LIN {X 0,Y 524.038,Z 318.828,A -85,B 0,C 180,E1 -4863.075,E2 -4863.075} C_VEL
LIN {X 0,Y 524.003,Z 318.833,A -85,B 0,C 180,E1 -4866.16,E2 -4866.16} C_VEL
LIN {X 0,Y 523.983,Z 318.838,A -85,B 0,C 180,E1 -4869.262,E2 -4869.262} C_VEL
LIN {X 0,Y 524.003,Z 318.838,A -85,B 0,C 180,E1 -4871.736,E2 -4871.736} C_VEL
LIN {X 0,Y 523.989,Z 318.836,A -85,B 0,C 180,E1 -4875.048,E2 -4875.048} C_VEL
LIN {X 0,Y 523.917,Z 318.849,A -85,B 0,C 180,E1 -4877.971,E2 -4877.971} C_VEL
LIN {X 0,Y 523.92,Z 318.841,A -85,B 0,C 180,E1 -4880.412,E2 -4880.412} C_VEL
LIN {X 0,Y 523.889,Z 318.848,A -85,B 0,C 180,E1 -4882.895,E2 -4882.895} C_VEL
LIN {X 0,Y 523.902,Z 318.85,A -85,B 0,C 180,E1 -4885.422,E2 -4885.422} C_VEL
LIN {X 0,Y 523.9,Z 318.847,A -85,B 0,C 180,E1 -4888.003,E2 -4888.003} C_VEL
LIN {X 0,Y 523.901,Z 318.839,A -85,B 0,C 180,E1 -4890.846,E2 -4890.846} C_VEL
LIN {X 0,Y 523.929,Z 318.847,A -85,B 0,C 180,E1 -4893.729,E2 -4893.729} C_VEL
LIN {X 0,Y 523.861,Z 318.844,A -85,B 0,C 180,E1 -4896.394,E2 -4896.394} C_VEL
LIN {X 0,Y 523.889,Z 318.852,A -85,B 0,C 180,E1 -4899.088,E2 -4899.088} C_VEL
LIN {X 0,Y 523.889,Z 318.848,A -85,B 0,C 180,E1 -4902.126,E2 -4902.126} C_VEL
LIN {X 0,Y 523.931,Z 318.847,A -85,B 0,C 180,E1 -4905.312,E2 -4905.312} C_VEL
LIN {X 0,Y 523.872,Z 318.851,A -85,B 0,C 180,E1 -4906.869,E2 -4906.869} C_VEL
LIN {X 0,Y 523.182,Z 318.943,A -85,B 0,C 180,E1 -4907.51,E2 -4907.51} C_VEL
LIN {X 0,Y 520.313,Z 319.296,A -85,B 0,C 180,E1 -4908.552,E2 -4908.552} C_VEL
LIN {X 0,Y 517.911,Z 319.598,A -85,B 0,C 180,E1 -4909.39,E2 -4909.39} C_VEL
LIN {X 0,Y 516.897,Z 319.721,A -85,B 0,C 180,E1 -4910.038,E2 -4910.038} C_VEL
LIN {X 0,Y 516.823,Z 319.729,A -85,B 0,C 180,E1 -4910.257,E2 -4910.257} C_VEL
LIN {X 0,Y 516.799,Z 319.74,A -85,B 0,C 180,E1 -4913.247,E2 -4913.247} C_VEL
LIN {X 0,Y 516.869,Z 319.723,A -85,B 0,C 180,E1 -4916.117,E2 -4916.117} C_VEL
LIN {X 0,Y 516.852,Z 319.731,A -85,B 0,C 180,E1 -4918.944,E2 -4918.944} C_VEL
LIN {X 0,Y 516.878,Z 319.819,A -85,B 0,C 180,E1 -4922.214,E2 -4922.214} C_VEL
LIN {X 0,Y 518.337,Z 327.517,A -85,B 0,C 180,E1 -4923.638,E2 -4923.638} C_VEL
LIN {X 0,Y 517.957,Z 343.652,A -85,B 0,C 180,E1 -4926.406,E2 -4926.406} C_VEL
LIN {X 0,Y 518.607,Z 346.948,A -85,B 0,C 180,E1 -4926.504,E2 -4926.504} C_VEL
LIN {X 0,Y 520.476,Z 356.835,A -85,B 0,C 180,E1 -4926.715,E2 -4926.715} C_VEL
LIN {X 0,Y 519.751,Z 479.979,A -85,B 0,C 180,E1 -4928.457,E2 -4928.457} C_VEL
LIN {X 0,Y 519.484,Z 494.208,A -85,B 0,C 180,E1 -4928.809,E2 -4928.809} C_VEL
LIN {X 0,Y 519.165,Z 508.132,A -85,B 0,C 180,E1 -4929.319,E2 -4929.319} C_VEL
LIN {X 0,Y 518.806,Z 521.885,A -85,B 0,C 180,E1 -4929.998,E2 -4929.998} C_VEL
LIN {X 0,Y 518.35,Z 534.66,A -85,B 0,C 180,E1 -4930.804,E2 -4930.804} C_VEL
LIN {X 0,Y 517.995,Z 545.305,A -85,B 0,C 180,E1 -4931.633,E2 -4931.633} C_VEL
LIN {X 0,Y 517.56,Z 555.862,A -85,B 0,C 180,E1 -4932.618,E2 -4932.618} C_VEL
LIN {X 0,Y 517.214,Z 566.524,A -85,B 0,C 180,E1 -4933.826,E2 -4933.826} C_VEL
LIN {X 0,Y 516.89,Z 575.271,A -85,B 0,C 180,E1 -4935.028,E2 -4935.028} C_VEL
LIN {X 0,Y 516.643,Z 583.607,A -85,B 0,C 180,E1 -4936.429,E2 -4936.429} C_VEL
LIN {X 0,Y 516.481,Z 590.258,A -85,B 0,C 180,E1 -4937.824,E2 -4937.824} C_VEL
LIN {X 0,Y 516.386,Z 594.836,A -85,B 0,C 180,E1 -4939.016,E2 -4939.016} C_VEL
LIN {X 0,Y 516.303,Z 598.458,A -85,B 0,C 180,E1 -4940.203,E2 -4940.203} C_VEL
LIN {X 0,Y 516.257,Z 601.259,A -85,B 0,C 180,E1 -4941.388,E2 -4941.388} C_VEL
LIN {X 0,Y 516.284,Z 603.699,A -85,B 0,C 180,E1 -4942.963,E2 -4942.963} C_VEL
LIN {X 0,Y 516.271,Z 604.789,A -85,B 0,C 180,E1 -4944.532,E2 -4944.532} C_VEL
LIN {X 0,Y 516.293,Z 604.557,A -85,B 0,C 180,E1 -4946.097,E2 -4946.097} C_VEL
LIN {X 0,Y 516.259,Z 603.009,A -85,B 0,C 180,E1 -4947.659,E2 -4947.659} C_VEL
LIN {X 0,Y 516.172,Z 600.122,A -85,B 0,C 180,E1 -4949.22,E2 -4949.22} C_VEL
LIN {X 0,Y 516.248,Z 595.813,A -85,B 0,C 180,E1 -4950.78,E2 -4950.78} C_VEL
LIN {X 0,Y 516.372,Z 589.959,A -85,B 0,C 180,E1 -4952.34,E2 -4952.34} C_VEL
LIN {X 0,Y 516.636,Z 583.37,A -85,B 0,C 180,E1 -4953.705,E2 -4953.705} C_VEL
LIN {X 0,Y 516.969,Z 575.193,A -85,B 0,C 180,E1 -4955.07,E2 -4955.07} C_VEL
LIN {X 0,Y 517.262,Z 566.698,A -85,B 0,C 180,E1 -4956.24,E2 -4956.24} C_VEL
LIN {X 0,Y 517.567,Z 556.458,A -85,B 0,C 180,E1 -4957.409,E2 -4957.409} C_VEL
LIN {X 0,Y 517.997,Z 544.966,A -85,B 0,C 180,E1 -4958.485,E2 -4958.485} C_VEL
LIN {X 0,Y 518.378,Z 533.526,A -85,B 0,C 180,E1 -4959.363,E2 -4959.363} C_VEL
LIN {X 0,Y 518.787,Z 520.975,A -85,B 0,C 180,E1 -4960.143,E2 -4960.143} C_VEL
LIN {X 0,Y 519.171,Z 507.994,A -85,B 0,C 180,E1 -4960.777,E2 -4960.777} C_VEL
LIN {X 0,Y 519.532,Z 493.96,A -85,B 0,C 180,E1 -4961.287,E2 -4961.287} C_VEL
LIN {X 0,Y 519.706,Z 480.239,A -85,B 0,C 180,E1 -4961.629,E2 -4961.629} C_VEL
LIN {X 0,Y 520.413,Z 355.748,A -85,B 0,C 180,E1 -4963.392,E2 -4963.392} C_VEL
LIN {X 0,Y 517.973,Z 343.725,A -85,B 0,C 180,E1 -4963.666,E2 -4963.666} C_VEL
LIN {X 0,Y 518.387,Z 328.115,A -85,B 0,C 180,E1 -4966.339,E2 -4966.339} C_VEL
LIN {X 0,Y 517.157,Z 321.108,A -85,B 0,C 180,E1 -4967.626,E2 -4967.626} C_VEL
LIN {X 0,Y 516.889,Z 319.725,A -85,B 0,C 180,E1 -4967.934,E2 -4967.934} C_VEL
LIN {X 0,Y 516.881,Z 319.729,A -85,B 0,C 180,E1 -4970.703,E2 -4970.703} C_VEL
LIN {X 0,Y 516.853,Z 319.73,A -85,B 0,C 180,E1 -4973.225,E2 -4973.225} C_VEL
LIN {X 0,Y 516.858,Z 319.726,A -85,B 0,C 180,E1 -4976.176,E2 -4976.176} C_VEL
LIN {X 0,Y 516.831,Z 319.731,A -85,B 0,C 180,E1 -4978.421,E2 -4978.421} C_VEL
LIN {X 0,Y 516.851,Z 319.73,A -85,B 0,C 180,E1 -4981.112,E2 -4981.112} C_VEL
LIN {X 0,Y 516.868,Z 319.723,A -85,B 0,C 180,E1 -4983.958,E2 -4983.958} C_VEL
LIN {X 0,Y 516.799,Z 319.738,A -85,B 0,C 180,E1 -4986.753,E2 -4986.753} C_VEL
LIN {X 0,Y 516.831,Z 319.726,A -85,B 0,C 180,E1 -4989.726,E2 -4989.726} C_VEL
LIN {X 0,Y 516.84,Z 319.732,A -85,B 0,C 180,E1 -4992.836,E2 -4992.836} C_VEL
LIN {X 0,Y 516.9,Z 319.721,A -85,B 0,C 180,E1 -4995.007,E2 -4995.007} C_VEL
LIN {X 0,Y 516.833,Z 319.732,A -85,B 0,C 180,E1 -4998.409,E2 -4998.409} C_VEL
LIN {X 0,Y 516.856,Z 319.724,A -85,B 0,C 180,E1 -5001.281,E2 -5001.281} C_VEL
LIN {X 0,Y 516.853,Z 319.731,A -85,B 0,C 180,E1 -5004.673,E2 -5004.673} C_VEL
LIN {X 0,Y 516.871,Z 319.718,A -85,B 0,C 180,E1 -5007.462,E2 -5007.462} C_VEL
LIN {X 0,Y 516.848,Z 319.732,A -85,B 0,C 180,E1 -5010.49,E2 -5010.49} C_VEL
LIN {X 0,Y 516.84,Z 319.723,A -85,B 0,C 180,E1 -5013.337,E2 -5013.337} C_VEL
LIN {X 0,Y 516.884,Z 319.723,A -85,B 0,C 180,E1 -5015.926,E2 -5015.926} C_VEL
LIN {X 0,Y 516.869,Z 319.721,A -85,B 0,C 180,E1 -5018.461,E2 -5018.461} C_VEL
LIN {X 0,Y 516.883,Z 319.717,A -85,B 0,C 180,E1 -5020.954,E2 -5020.954} C_VEL
LIN {X 0,Y 516.835,Z 319.726,A -85,B 0,C 180,E1 -5023.407,E2 -5023.407} C_VEL
LIN {X 0,Y 516.877,Z 319.723,A -85,B 0,C 180,E1 -5025.833,E2 -5025.833} C_VEL
LIN {X 0,Y 516.952,Z 319.702,A -85,B 0,C 180,E1 -5029.028,E2 -5029.028} C_VEL
LIN {X 0,Y 516.947,Z 319.718,A -85,B 0,C 180,E1 -5032.186,E2 -5032.186} C_VEL
LIN {X 0,Y 516.991,Z 319.71,A -85,B 0,C 180,E1 -5034.539,E2 -5034.539} C_VEL
LIN {X 0,Y 517.081,Z 319.697,A -85,B 0,C 180,E1 -5037.663,E2 -5037.663} C_VEL
LIN {X 0,Y 517.093,Z 319.692,A -85,B 0,C 180,E1 -5040.779,E2 -5040.779} C_VEL
LIN {X 0,Y 516.951,Z 319.711,A -85,B 0,C 180,E1 -5043.117,E2 -5043.117} C_VEL
LIN {X 0,Y 516.978,Z 319.713,A -85,B 0,C 180,E1 -5046.243,E2 -5046.243} C_VEL
LIN {X 0,Y 516.941,Z 319.714,A -85,B 0,C 180,E1 -5049.389,E2 -5049.389} C_VEL
LIN {X 0,Y 516.956,Z 319.717,A -85,B 0,C 180,E1 -5051.807,E2 -5051.807} C_VEL
LIN {X 0,Y 516.949,Z 319.711,A -85,B 0,C 180,E1 -5055.146,E2 -5055.146} C_VEL
LIN {X 0,Y 516.916,Z 319.719,A -85,B 0,C 180,E1 -5058.222,E2 -5058.222} C_VEL
LIN {X 0,Y 516.916,Z 319.716,A -85,B 0,C 180,E1 -5060.701,E2 -5060.701} C_VEL
LIN {X 0,Y 516.893,Z 319.724,A -85,B 0,C 180,E1 -5064.073,E2 -5064.073} C_VEL
LIN {X 0,Y 516.914,Z 319.716,A -85,B 0,C 180,E1 -5066.658,E2 -5066.658} C_VEL
LIN {X 0,Y 516.913,Z 319.722,A -85,B 0,C 180,E1 -5069.523,E2 -5069.523} C_VEL
LIN {X 0,Y 516.898,Z 319.718,A -85,B 0,C 180,E1 -5072.543,E2 -5072.543} C_VEL
LIN {X 0,Y 516.871,Z 319.727,A -85,B 0,C 180,E1 -5075.33,E2 -5075.33} C_VEL
LIN {X 0,Y 516.881,Z 319.725,A -85,B 0,C 180,E1 -5077.943,E2 -5077.943} C_VEL
LIN {X 0,Y 516.885,Z 319.721,A -85,B 0,C 180,E1 -5080.741,E2 -5080.741} C_VEL
LIN {X 0,Y 516.884,Z 319.721,A -85,B 0,C 180,E1 -5082.831,E2 -5082.831} C_VEL
LIN {X 0,Y 516.897,Z 319.721,A -85,B 0,C 180,E1 -5085.007,E2 -5085.007} C_VEL
LIN {X 0,Y 516.915,Z 319.717,A -85,B 0,C 180,E1 -5088.399,E2 -5088.399} C_VEL
LIN {X 0,Y 516.882,Z 319.728,A -85,B 0,C 180,E1 -5091.284,E2 -5091.284} C_VEL
LIN {X 0,Y 516.89,Z 319.722,A -85,B 0,C 180,E1 -5094.221,E2 -5094.221} C_VEL
LIN {X 0,Y 516.897,Z 319.725,A -85,B 0,C 180,E1 -5097.053,E2 -5097.053} C_VEL
LIN {X 0,Y 516.894,Z 319.724,A -85,B 0,C 180,E1 -5099.796,E2 -5099.796} C_VEL
LIN {X 0,Y 516.928,Z 319.718,A -85,B 0,C 180,E1 -5102.467,E2 -5102.467} C_VEL
LIN {X 0,Y 516.962,Z 319.819,A -85,B 0,C 180,E1 -5103.83,E2 -5103.83} C_VEL
LIN {X 0,Y 519.173,Z 330.998,A -85,B 0,C 180,E1 -5105.614,E2 -5105.614} C_VEL
LIN {X 0,Y 518.581,Z 350.939,A -85,B 0,C 180,E1 -5108.536,E2 -5108.536} C_VEL
LIN {X 0,Y 518.001,Z 370.708,A -85,B 0,C 180,E1 -5111.377,E2 -5111.377} C_VEL
LIN {X 0,Y 520.347,Z 384.922,A -85,B 0,C 180,E1 -5111.666,E2 -5111.666} C_VEL
LIN {X 0,Y 519.63,Z 509.015,A -85,B 0,C 180,E1 -5113.424,E2 -5113.424} C_VEL
LIN {X 0,Y 519.367,Z 523.324,A -85,B 0,C 180,E1 -5113.786,E2 -5113.786} C_VEL
LIN {X 0,Y 519.051,Z 536.906,A -85,B 0,C 180,E1 -5114.288,E2 -5114.288} C_VEL
LIN {X 0,Y 518.654,Z 550.881,A -85,B 0,C 180,E1 -5114.98,E2 -5114.98} C_VEL
LIN {X 0,Y 518.219,Z 563.384,A -85,B 0,C 180,E1 -5115.77,E2 -5115.77} C_VEL
LIN {X 0,Y 517.825,Z 574.814,A -85,B 0,C 180,E1 -5116.66,E2 -5116.66} C_VEL
LIN {X 0,Y 517.445,Z 585.278,A -85,B 0,C 180,E1 -5117.644,E2 -5117.644} C_VEL
LIN {X 0,Y 517.138,Z 595.771,A -85,B 0,C 180,E1 -5118.833,E2 -5118.833} C_VEL
LIN {X 0,Y 516.813,Z 604.395,A -85,B 0,C 180,E1 -5120.015,E2 -5120.015} C_VEL
LIN {X 0,Y 516.59,Z 612.657,A -85,B 0,C 180,E1 -5121.393,E2 -5121.393} C_VEL
LIN {X 0,Y 516.445,Z 618.44,A -85,B 0,C 180,E1 -5122.572,E2 -5122.572} C_VEL
LIN {X 0,Y 516.395,Z 623.18,A -85,B 0,C 180,E1 -5123.749,E2 -5123.749} C_VEL
LIN {X 0,Y 516.306,Z 627.019,A -85,B 0,C 180,E1 -5124.924,E2 -5124.924} C_VEL
LIN {X 0,Y 516.324,Z 629.978,A -85,B 0,C 180,E1 -5126.098,E2 -5126.098} C_VEL
LIN {X 0,Y 516.259,Z 632.685,A -85,B 0,C 180,E1 -5127.659,E2 -5127.659} C_VEL
LIN {X 0,Y 516.157,Z 634.024,A -85,B 0,C 180,E1 -5129.22,E2 -5129.22} C_VEL
LIN {X 0,Y 516.157,Z 634.024,A -85,B 0,C 180,E1 -5130.78,E2 -5130.78} C_VEL
LIN {X 0,Y 516.259,Z 632.686,A -85,B 0,C 180,E1 -5132.341,E2 -5132.341} C_VEL
LIN {X 0,Y 516.324,Z 629.98,A -85,B 0,C 180,E1 -5133.903,E2 -5133.903} C_VEL
LIN {X 0,Y 516.367,Z 625.828,A -85,B 0,C 180,E1 -5135.467,E2 -5135.467} C_VEL
LIN {X 0,Y 516.402,Z 620.109,A -85,B 0,C 180,E1 -5137.036,E2 -5137.036} C_VEL
LIN {X 0,Y 516.582,Z 613.665,A -85,B 0,C 180,E1 -5138.41,E2 -5138.41} C_VEL
LIN {X 0,Y 516.779,Z 605.659,A -85,B 0,C 180,E1 -5139.788,E2 -5139.788} C_VEL
LIN {X 0,Y 517.078,Z 597.288,A -85,B 0,C 180,E1 -5140.969,E2 -5140.969} C_VEL
LIN {X 0,Y 517.414,Z 586.88,A -85,B 0,C 180,E1 -5142.19,E2 -5142.19} C_VEL
LIN {X 0,Y 517.783,Z 575.973,A -85,B 0,C 180,E1 -5143.241,E2 -5143.241} C_VEL
LIN {X 0,Y 518.211,Z 563.369,A -85,B 0,C 180,E1 -5144.23,E2 -5144.23} C_VEL
LIN {X 0,Y 518.664,Z 550.862,A -85,B 0,C 180,E1 -5145.02,E2 -5145.02} C_VEL
LIN {X 0,Y 519.03,Z 538.006,A -85,B 0,C 180,E1 -5145.662,E2 -5145.662} C_VEL
LIN {X 0,Y 519.34,Z 524.353,A -85,B 0,C 180,E1 -5146.179,E2 -5146.179} C_VEL
LIN {X 0,Y 519.621,Z 510.128,A -85,B 0,C 180,E1 -5146.552,E2 -5146.552} C_VEL
LIN {X 0,Y 519.826,Z 481.992,A -85,B 0,C 180,E1 -5146.975,E2 -5146.975} C_VEL
LIN {X 0,Y 520.36,Z 383.971,A -85,B 0,C 180,E1 -5148.347,E2 -5148.347} C_VEL
LIN {X 0,Y 518.017,Z 370.538,A -85,B 0,C 180,E1 -5148.633,E2 -5148.633} C_VEL
LIN {X 0,Y 518.626,Z 349.478,A -85,B 0,C 180,E1 -5151.671,E2 -5151.671} C_VEL
LIN {X 0,Y 519.184,Z 330.985,A -85,B 0,C 180,E1 -5154.385,E2 -5154.385} C_VEL
LIN {X 0,Y 516.944,Z 319.769,A -85,B 0,C 180,E1 -5156.196,E2 -5156.196} C_VEL
LIN {X 0,Y 516.924,Z 319.717,A -85,B 0,C 180,E1 -5159.305,E2 -5159.305} C_VEL
LIN {X 0,Y 516.898,Z 319.725,A -85,B 0,C 180,E1 -5162.544,E2 -5162.544} C_VEL
LIN {X 0,Y 516.869,Z 319.724,A -85,B 0,C 180,E1 -5165.33,E2 -5165.33} C_VEL
LIN {X 0,Y 516.882,Z 319.723,A -85,B 0,C 180,E1 -5167.943,E2 -5167.943} C_VEL
LIN {X 0,Y 516.885,Z 319.725,A -85,B 0,C 180,E1 -5170.742,E2 -5170.742} C_VEL
LIN {X 0,Y 516.884,Z 319.723,A -85,B 0,C 180,E1 -5172.832,E2 -5172.832} C_VEL
LIN {X 0,Y 516.897,Z 319.72,A -85,B 0,C 180,E1 -5175.007,E2 -5175.007} C_VEL
LIN {X 0,Y 516.916,Z 319.723,A -85,B 0,C 180,E1 -5178.399,E2 -5178.399} C_VEL
LIN {X 0,Y 516.881,Z 319.72,A -85,B 0,C 180,E1 -5181.284,E2 -5181.284} C_VEL
LIN {X 0,Y 516.87,Z 319.727,A -85,B 0,C 180,E1 -5184.22,E2 -5184.22} C_VEL
LIN {X 0,Y 516.898,Z 319.718,A -85,B 0,C 180,E1 -5187.053,E2 -5187.053} C_VEL
LIN {X 0,Y 516.895,Z 319.721,A -85,B 0,C 180,E1 -5189.797,E2 -5189.797} C_VEL
LIN {X 0,Y 516.895,Z 319.723,A -85,B 0,C 180,E1 -5192.466,E2 -5192.466} C_VEL
LIN {X 0,Y 516.868,Z 319.722,A -85,B 0,C 180,E1 -5195.07,E2 -5195.07} C_VEL
LIN {X 0,Y 516.873,Z 319.722,A -85,B 0,C 180,E1 -5197.622,E2 -5197.622} C_VEL
LIN {X 0,Y 516.933,Z 319.723,A -85,B 0,C 180,E1 -5200.13,E2 -5200.13} C_VEL
LIN {X 0,Y 516.901,Z 319.719,A -85,B 0,C 180,E1 -5202.595,E2 -5202.595} C_VEL
LIN {X 0,Y 516.947,Z 319.712,A -85,B 0,C 180,E1 -5205.03,E2 -5205.03} C_VEL
LIN {X 0,Y 516.971,Z 319.715,A -85,B 0,C 180,E1 -5208.234,E2 -5208.234} C_VEL
LIN {X 0,Y 516.955,Z 319.711,A -85,B 0,C 180,E1 -5211.4,E2 -5211.4} C_VEL
LIN {X 0,Y 517.016,Z 319.705,A -85,B 0,C 180,E1 -5214.54,E2 -5214.54} C_VEL
LIN {X 0,Y 517.078,Z 319.697,A -85,B 0,C 180,E1 -5217.663,E2 -5217.663} C_VEL
LIN {X 0,Y 517.069,Z 319.703,A -85,B 0,C 180,E1 -5220,E2 -5220} C_VEL
LIN {X 0,Y 517.081,Z 319.697,A -85,B 0,C 180,E1 -5222.337,E2 -5222.337} C_VEL
LIN {X 0,Y 516.97,Z 319.708,A -85,B 0,C 180,E1 -5226.244,E2 -5226.244} C_VEL
LIN {X 0,Y 516.939,Z 319.717,A -85,B 0,C 180,E1 -5229.39,E2 -5229.39} C_VEL
LIN {X 0,Y 516.957,Z 319.716,A -85,B 0,C 180,E1 -5231.807,E2 -5231.807} C_VEL
LIN {X 0,Y 516.942,Z 319.715,A -85,B 0,C 180,E1 -5235.143,E2 -5235.143} C_VEL
LIN {X 0,Y 516.878,Z 319.723,A -85,B 0,C 180,E1 -5238.224,E2 -5238.224} C_VEL
LIN {X 0,Y 516.875,Z 319.718,A -85,B 0,C 180,E1 -5240.703,E2 -5240.703} C_VEL
LIN {X 0,Y 516.844,Z 319.729,A -85,B 0,C 180,E1 -5243.225,E2 -5243.225} C_VEL
LIN {X 0,Y 516.883,Z 319.722,A -85,B 0,C 180,E1 -5246.181,E2 -5246.181} C_VEL
LIN {X 0,Y 516.833,Z 319.724,A -85,B 0,C 180,E1 -5248.421,E2 -5248.421} C_VEL
LIN {X 0,Y 516.852,Z 319.719,A -85,B 0,C 180,E1 -5251.112,E2 -5251.112} C_VEL
LIN {X 0,Y 516.884,Z 319.722,A -85,B 0,C 180,E1 -5253.961,E2 -5253.961} C_VEL
LIN {X 0,Y 516.803,Z 319.724,A -85,B 0,C 180,E1 -5256.753,E2 -5256.753} C_VEL
LIN {X 0,Y 516.856,Z 319.729,A -85,B 0,C 180,E1 -5259.189,E2 -5259.189} C_VEL
LIN {X 0,Y 516.834,Z 319.729,A -85,B 0,C 180,E1 -5261.783,E2 -5261.783} C_VEL
LIN {X 0,Y 516.9,Z 319.723,A -85,B 0,C 180,E1 -5265.007,E2 -5265.007} C_VEL
LIN {X 0,Y 516.83,Z 319.729,A -85,B 0,C 180,E1 -5268.41,E2 -5268.41} C_VEL
LIN {X 0,Y 516.823,Z 319.729,A -85,B 0,C 180,E1 -5270.257,E2 -5270.257} C_VEL
LIN {X 0,Y 516.178,Z 319.815,A -85,B 0,C 180,E1 -5270.907,E2 -5270.907} C_VEL
LIN {X 0,Y 513.324,Z 320.171,A -85,B 0,C 180,E1 -5271.963,E2 -5271.963} C_VEL
LIN {X 0,Y 510.894,Z 320.475,A -85,B 0,C 180,E1 -5272.813,E2 -5272.813} C_VEL
LIN {X 0,Y 509.846,Z 320.604,A -85,B 0,C 180,E1 -5273.47,E2 -5273.47} C_VEL
LIN {X 0,Y 509.758,Z 320.612,A -85,B 0,C 180,E1 -5273.692,E2 -5273.692} C_VEL
LIN {X 0,Y 509.827,Z 320.601,A -85,B 0,C 180,E1 -5276.536,E2 -5276.536} C_VEL
LIN {X 0,Y 509.804,Z 320.609,A -85,B 0,C 180,E1 -5279.331,E2 -5279.331} C_VEL
LIN {X 0,Y 509.835,Z 320.687,A -85,B 0,C 180,E1 -5281.998,E2 -5281.998} C_VEL
LIN {X 0,Y 511.465,Z 329.337,A -85,B 0,C 180,E1 -5283.625,E2 -5283.625} C_VEL
LIN {X 0,Y 511.046,Z 343.971,A -85,B 0,C 180,E1 -5286.167,E2 -5286.167} C_VEL
LIN {X 0,Y 513.649,Z 356.408,A -85,B 0,C 180,E1 -5286.453,E2 -5286.453} C_VEL
LIN {X 0,Y 512.97,Z 480.449,A -85,B 0,C 180,E1 -5288.237,E2 -5288.237} C_VEL
LIN {X 0,Y 512.669,Z 494.537,A -85,B 0,C 180,E1 -5288.592,E2 -5288.592} C_VEL
LIN {X 0,Y 512.329,Z 508.352,A -85,B 0,C 180,E1 -5289.105,E2 -5289.105} C_VEL
LIN {X 0,Y 511.937,Z 520.818,A -85,B 0,C 180,E1 -5289.718,E2 -5289.718} C_VEL
LIN {X 0,Y 511.522,Z 533.849,A -85,B 0,C 180,E1 -5290.538,E2 -5290.538} C_VEL
LIN {X 0,Y 511.067,Z 545.623,A -85,B 0,C 180,E1 -5291.457,E2 -5291.457} C_VEL
LIN {X 0,Y 510.57,Z 557.352,A -85,B 0,C 180,E1 -5292.579,E2 -5292.579} C_VEL
LIN {X 0,Y 510.204,Z 567.776,A -85,B 0,C 180,E1 -5293.803,E2 -5293.803} C_VEL
LIN {X 0,Y 509.839,Z 576.337,A -85,B 0,C 180,E1 -5295.021,E2 -5295.021} C_VEL
LIN {X 0,Y 509.566,Z 584.47,A -85,B 0,C 180,E1 -5296.44,E2 -5296.44} C_VEL
LIN {X 0,Y 509.42,Z 590.175,A -85,B 0,C 180,E1 -5297.652,E2 -5297.652} C_VEL
LIN {X 0,Y 509.285,Z 596.116,A -85,B 0,C 180,E1 -5299.263,E2 -5299.263} C_VEL
LIN {X 0,Y 509.178,Z 599.541,A -85,B 0,C 180,E1 -5300.466,E2 -5300.466} C_VEL
LIN {X 0,Y 509.17,Z 602.756,A -85,B 0,C 180,E1 -5302.066,E2 -5302.066} C_VEL
LIN {X 0,Y 509.174,Z 604.57,A -85,B 0,C 180,E1 -5303.66,E2 -5303.66} C_VEL
LIN {X 0,Y 509.128,Z 605.055,A -85,B 0,C 180,E1 -5305.249,E2 -5305.249} C_VEL
LIN {X 0,Y 509.182,Z 604.219,A -85,B 0,C 180,E1 -5306.835,E2 -5306.835} C_VEL
LIN {X 0,Y 509.116,Z 602.063,A -85,B 0,C 180,E1 -5308.418,E2 -5308.418} C_VEL
LIN {X 0,Y 509.13,Z 598.535,A -85,B 0,C 180,E1 -5310,E2 -5310} C_VEL
LIN {X 0,Y 509.303,Z 594.935,A -85,B 0,C 180,E1 -5311.186,E2 -5311.186} C_VEL
LIN {X 0,Y 509.302,Z 590.439,A -85,B 0,C 180,E1 -5312.373,E2 -5312.373} C_VEL
LIN {X 0,Y 509.586,Z 583.925,A -85,B 0,C 180,E1 -5313.756,E2 -5313.756} C_VEL
LIN {X 0,Y 509.95,Z 575.857,A -85,B 0,C 180,E1 -5315.14,E2 -5315.14} C_VEL
LIN {X 0,Y 510.264,Z 567.451,A -85,B 0,C 180,E1 -5316.326,E2 -5316.326} C_VEL
LIN {X 0,Y 510.585,Z 557.063,A -85,B 0,C 180,E1 -5317.539,E2 -5317.539} C_VEL
LIN {X 0,Y 511.048,Z 545.971,A -85,B 0,C 180,E1 -5318.601,E2 -5318.601} C_VEL
LIN {X 0,Y 511.51,Z 533.299,A -85,B 0,C 180,E1 -5319.59,E2 -5319.59} C_VEL
LIN {X 0,Y 511.951,Z 520.646,A -85,B 0,C 180,E1 -5320.38,E2 -5320.38} C_VEL
LIN {X 0,Y 512.322,Z 507.526,A -85,B 0,C 180,E1 -5321.022,E2 -5321.022} C_VEL
LIN {X 0,Y 512.72,Z 493.202,A -85,B 0,C 180,E1 -5321.539,E2 -5321.539} C_VEL
LIN {X 0,Y 512.957,Z 478.712,A -85,B 0,C 180,E1 -5321.885,E2 -5321.885} C_VEL
LIN {X 0,Y 513.628,Z 356.48,A -85,B 0,C 180,E1 -5323.636,E2 -5323.636} C_VEL
LIN {X 0,Y 511.049,Z 343.927,A -85,B 0,C 180,E1 -5323.926,E2 -5323.926} C_VEL
LIN {X 0,Y 511.479,Z 329.875,A -85,B 0,C 180,E1 -5326.361,E2 -5326.361} C_VEL
LIN {X 0,Y 510.552,Z 324.126,A -85,B 0,C 180,E1 -5327.422,E2 -5327.422} C_VEL
LIN {X 0,Y 509.848,Z 320.603,A -85,B 0,C 180,E1 -5328.099,E2 -5328.099} C_VEL
LIN {X 0,Y 509.827,Z 320.608,A -85,B 0,C 180,E1 -5331.003,E2 -5331.003} C_VEL
LIN {X 0,Y 509.811,Z 320.604,A -85,B 0,C 180,E1 -5333.565,E2 -5333.565} C_VEL
LIN {X 0,Y 509.799,Z 320.607,A -85,B 0,C 180,E1 -5336.352,E2 -5336.352} C_VEL
LIN {X 0,Y 509.795,Z 320.612,A -85,B 0,C 180,E1 -5338.85,E2 -5338.85} C_VEL
LIN {X 0,Y 509.79,Z 320.605,A -85,B 0,C 180,E1 -5341.592,E2 -5341.592} C_VEL
LIN {X 0,Y 509.822,Z 320.604,A -85,B 0,C 180,E1 -5344.416,E2 -5344.416} C_VEL
LIN {X 0,Y 509.762,Z 320.609,A -85,B 0,C 180,E1 -5347.346,E2 -5347.346} C_VEL
LIN {X 0,Y 509.79,Z 320.608,A -85,B 0,C 180,E1 -5350.387,E2 -5350.387} C_VEL
LIN {X 0,Y 509.794,Z 320.603,A -85,B 0,C 180,E1 -5353.575,E2 -5353.575} C_VEL
LIN {X 0,Y 509.794,Z 320.608,A -85,B 0,C 180,E1 -5356.425,E2 -5356.425} C_VEL
LIN {X 0,Y 509.789,Z 320.603,A -85,B 0,C 180,E1 -5359.613,E2 -5359.613} C_VEL
LIN {X 0,Y 509.776,Z 320.611,A -85,B 0,C 180,E1 -5362.655,E2 -5362.655} C_VEL
LIN {X 0,Y 509.842,Z 320.598,A -85,B 0,C 180,E1 -5365.8,E2 -5365.8} C_VEL
LIN {X 0,Y 509.819,Z 320.605,A -85,B 0,C 180,E1 -5368.726,E2 -5368.726} C_VEL
LIN {X 0,Y 509.826,Z 320.601,A -85,B 0,C 180,E1 -5372.05,E2 -5372.05} C_VEL
LIN {X 0,Y 509.804,Z 320.607,A -85,B 0,C 180,E1 -5374.7,E2 -5374.7} C_VEL
LIN {X 0,Y 509.827,Z 320.597,A -85,B 0,C 180,E1 -5377.459,E2 -5377.459} C_VEL
LIN {X 0,Y 509.893,Z 320.584,A -85,B 0,C 180,E1 -5379.843,E2 -5379.843} C_VEL
LIN {X 0,Y 509.85,Z 320.602,A -85,B 0,C 180,E1 -5382.346,E2 -5382.346} C_VEL
LIN {X 0,Y 509.888,Z 320.593,A -85,B 0,C 180,E1 -5384.818,E2 -5384.818} C_VEL
LIN {X 0,Y 509.906,Z 320.589,A -85,B 0,C 180,E1 -5388.124,E2 -5388.124} C_VEL
LIN {X 0,Y 509.904,Z 320.586,A -85,B 0,C 180,E1 -5391.279,E2 -5391.279} C_VEL
LIN {X 0,Y 509.946,Z 320.588,A -85,B 0,C 180,E1 -5394.464,E2 -5394.464} C_VEL
LIN {X 0,Y 510.051,Z 320.572,A -85,B 0,C 180,E1 -5397.631,E2 -5397.631} C_VEL
LIN {X 0,Y 510.042,Z 320.57,A -85,B 0,C 180,E1 -5400.789,E2 -5400.789} C_VEL
LIN {X 0,Y 509.896,Z 320.59,A -85,B 0,C 180,E1 -5403.16,E2 -5403.16} C_VEL
LIN {X 0,Y 509.925,Z 320.591,A -85,B 0,C 180,E1 -5406.33,E2 -5406.33} C_VEL
LIN {X 0,Y 509.882,Z 320.594,A -85,B 0,C 180,E1 -5409.52,E2 -5409.52} C_VEL
LIN {X 0,Y 509.908,Z 320.597,A -85,B 0,C 180,E1 -5411.931,E2 -5411.931} C_VEL
LIN {X 0,Y 509.898,Z 320.59,A -85,B 0,C 180,E1 -5415.241,E2 -5415.241} C_VEL
LIN {X 0,Y 509.861,Z 320.595,A -85,B 0,C 180,E1 -5418.484,E2 -5418.484} C_VEL
LIN {X 0,Y 509.854,Z 320.596,A -85,B 0,C 180,E1 -5421.001,E2 -5421.001} C_VEL
LIN {X 0,Y 509.825,Z 320.604,A -85,B 0,C 180,E1 -5423.564,E2 -5423.564} C_VEL
LIN {X 0,Y 509.909,Z 320.591,A -85,B 0,C 180,E1 -5426.377,E2 -5426.377} C_VEL
LIN {X 0,Y 509.86,Z 320.603,A -85,B 0,C 180,E1 -5429.751,E2 -5429.751} C_VEL
LIN {X 0,Y 509.876,Z 320.593,A -85,B 0,C 180,E1 -5432.774,E2 -5432.774} C_VEL
LIN {X 0,Y 509.83,Z 320.607,A -85,B 0,C 180,E1 -5435.578,E2 -5435.578} C_VEL
LIN {X 0,Y 509.851,Z 320.597,A -85,B 0,C 180,E1 -5438.338,E2 -5438.338} C_VEL
LIN {X 0,Y 509.857,Z 320.603,A -85,B 0,C 180,E1 -5441.425,E2 -5441.425} C_VEL
LIN {X 0,Y 509.841,Z 320.598,A -85,B 0,C 180,E1 -5444.67,E2 -5444.67} C_VEL
LIN {X 0,Y 509.857,Z 320.597,A -85,B 0,C 180,E1 -5448.103,E2 -5448.103} C_VEL
LIN {X 0,Y 509.847,Z 320.598,A -85,B 0,C 180,E1 -5450.647,E2 -5450.647} C_VEL
LIN {X 0,Y 509.836,Z 320.607,A -85,B 0,C 180,E1 -5453.648,E2 -5453.648} C_VEL
LIN {X 0,Y 509.863,Z 320.598,A -85,B 0,C 180,E1 -5456.539,E2 -5456.539} C_VEL
LIN {X 0,Y 509.847,Z 320.605,A -85,B 0,C 180,E1 -5459.334,E2 -5459.334} C_VEL
LIN {X 0,Y 509.894,Z 320.595,A -85,B 0,C 180,E1 -5462.054,E2 -5462.054} C_VEL
LIN {X 0,Y 509.917,Z 320.741,A -85,B 0,C 180,E1 -5463.621,E2 -5463.621} C_VEL
LIN {X 0,Y 512.276,Z 332.475,A -85,B 0,C 180,E1 -5465.521,E2 -5465.521} C_VEL
LIN {X 0,Y 511.648,Z 352.174,A -85,B 0,C 180,E1 -5468.442,E2 -5468.442} C_VEL
LIN {X 0,Y 511.076,Z 370.527,A -85,B 0,C 180,E1 -5471.116,E2 -5471.116} C_VEL
LIN {X 0,Y 513.603,Z 385.61,A -85,B 0,C 180,E1 -5471.429,E2 -5471.429} C_VEL
LIN {X 0,Y 512.831,Z 508.806,A -85,B 0,C 180,E1 -5473.197,E2 -5473.197} C_VEL
LIN {X 0,Y 512.524,Z 523.566,A -85,B 0,C 180,E1 -5473.579,E2 -5473.579} C_VEL
LIN {X 0,Y 512.163,Z 537.833,A -85,B 0,C 180,E1 -5474.122,E2 -5474.122} C_VEL
LIN {X 0,Y 511.77,Z 550.676,A -85,B 0,C 180,E1 -5474.773,E2 -5474.773} C_VEL
LIN {X 0,Y 511.299,Z 563.18,A -85,B 0,C 180,E1 -5475.574,E2 -5475.574} C_VEL
LIN {X 0,Y 510.865,Z 574.61,A -85,B 0,C 180,E1 -5476.475,E2 -5476.475} C_VEL
LIN {X 0,Y 510.451,Z 585.3,A -85,B 0,C 180,E1 -5477.495,E2 -5477.495} C_VEL
LIN {X 0,Y 510.122,Z 595.568,A -85,B 0,C 180,E1 -5478.678,E2 -5478.678} C_VEL
LIN {X 0,Y 509.754,Z 604.192,A -85,B 0,C 180,E1 -5479.876,E2 -5479.876} C_VEL
LIN {X 0,Y 509.536,Z 612.455,A -85,B 0,C 180,E1 -5481.273,E2 -5481.273} C_VEL
LIN {X 0,Y 509.369,Z 618.238,A -85,B 0,C 180,E1 -5482.468,E2 -5482.468} C_VEL
LIN {X 0,Y 509.304,Z 624.381,A -85,B 0,C 180,E1 -5484.06,E2 -5484.06} C_VEL
LIN {X 0,Y 509.181,Z 627.888,A -85,B 0,C 180,E1 -5485.25,E2 -5485.25} C_VEL
LIN {X 0,Y 509.193,Z 631.304,A -85,B 0,C 180,E1 -5486.835,E2 -5486.835} C_VEL
LIN {X 0,Y 509.109,Z 633.322,A -85,B 0,C 180,E1 -5488.418,E2 -5488.418} C_VEL
LIN {X 0,Y 509.064,Z 633.99,A -85,B 0,C 180,E1 -5490,E2 -5490} C_VEL
LIN {X 0,Y 509.109,Z 633.322,A -85,B 0,C 180,E1 -5491.582,E2 -5491.582} C_VEL
LIN {X 0,Y 509.193,Z 631.305,A -85,B 0,C 180,E1 -5493.165,E2 -5493.165} C_VEL
LIN {X 0,Y 509.181,Z 627.886,A -85,B 0,C 180,E1 -5494.75,E2 -5494.75} C_VEL
LIN {X 0,Y 509.303,Z 624.373,A -85,B 0,C 180,E1 -5495.94,E2 -5495.94} C_VEL
LIN {X 0,Y 509.327,Z 619.904,A -85,B 0,C 180,E1 -5497.134,E2 -5497.134} C_VEL
LIN {X 0,Y 509.523,Z 613.46,A -85,B 0,C 180,E1 -5498.527,E2 -5498.527} C_VEL
LIN {X 0,Y 509.73,Z 605.452,A -85,B 0,C 180,E1 -5499.924,E2 -5499.924} C_VEL
LIN {X 0,Y 510.048,Z 597.081,A -85,B 0,C 180,E1 -5501.123,E2 -5501.123} C_VEL
LIN {X 0,Y 510.412,Z 586.364,A -85,B 0,C 180,E1 -5502.394,E2 -5502.394} C_VEL
LIN {X 0,Y 510.819,Z 575.765,A -85,B 0,C 180,E1 -5503.425,E2 -5503.425} C_VEL
LIN {X 0,Y 511.232,Z 564.589,A -85,B 0,C 180,E1 -5504.327,E2 -5504.327} C_VEL
LIN {X 0,Y 511.688,Z 552.423,A -85,B 0,C 180,E1 -5505.127,E2 -5505.127} C_VEL
LIN {X 0,Y 512.138,Z 538.927,A -85,B 0,C 180,E1 -5505.828,E2 -5505.828} C_VEL
LIN {X 0,Y 512.511,Z 524.779,A -85,B 0,C 180,E1 -5506.38,E2 -5506.38} C_VEL
LIN {X 0,Y 512.802,Z 511.052,A -85,B 0,C 180,E1 -5506.752,E2 -5506.752} C_VEL
LIN {X 0,Y 512.968,Z 490.727,A -85,B 0,C 180,E1 -5507.08,E2 -5507.08} C_VEL
LIN {X 0,Y 513.646,Z 385.502,A -85,B 0,C 180,E1 -5508.57,E2 -5508.57} C_VEL
LIN {X 0,Y 511.075,Z 370.328,A -85,B 0,C 180,E1 -5508.896,E2 -5508.896} C_VEL
LIN {X 0,Y 511.724,Z 349.297,A -85,B 0,C 180,E1 -5511.978,E2 -5511.978} C_VEL
LIN {X 0,Y 512.292,Z 332.532,A -85,B 0,C 180,E1 -5514.48,E2 -5514.48} C_VEL
LIN {X 0,Y 510.289,Z 322.34,A -85,B 0,C 180,E1 -5516.15,E2 -5516.15} C_VEL
LIN {X 0,Y 509.909,Z 320.598,A -85,B 0,C 180,E1 -5516.486,E2 -5516.486} C_VEL
LIN {X 0,Y 509.878,Z 320.599,A -85,B 0,C 180,E1 -5518.844,E2 -5518.844} C_VEL
LIN {X 0,Y 509.822,Z 320.601,A -85,B 0,C 180,E1 -5521.59,E2 -5521.59} C_VEL
LIN {X 0,Y 509.85,Z 320.603,A -85,B 0,C 180,E1 -5524.414,E2 -5524.414} C_VEL
LIN {X 0,Y 509.818,Z 320.602,A -85,B 0,C 180,E1 -5527.341,E2 -5527.341} C_VEL
LIN {X 0,Y 509.84,Z 320.604,A -85,B 0,C 180,E1 -5530.382,E2 -5530.382} C_VEL
LIN {X 0,Y 509.824,Z 320.6,A -85,B 0,C 180,E1 -5533.062,E2 -5533.062} C_VEL
LIN {X 0,Y 509.824,Z 320.6,A -85,B 0,C 180,E1 -5535.794,E2 -5535.794} C_VEL
LIN {X 0,Y 509.858,Z 320.602,A -85,B 0,C 180,E1 -5538.575,E2 -5538.575} C_VEL
LIN {X 0,Y 509.852,Z 320.597,A -85,B 0,C 180,E1 -5541.787,E2 -5541.787} C_VEL
LIN {X 0,Y 509.83,Z 320.604,A -85,B 0,C 180,E1 -5544.622,E2 -5544.622} C_VEL
LIN {X 0,Y 509.864,Z 320.594,A -85,B 0,C 180,E1 -5547.481,E2 -5547.481} C_VEL
LIN {X 0,Y 509.862,Z 320.601,A -85,B 0,C 180,E1 -5550.274,E2 -5550.274} C_VEL
LIN {X 0,Y 509.877,Z 320.593,A -85,B 0,C 180,E1 -5553.63,E2 -5553.63} C_VEL
LIN {X 0,Y 509.825,Z 320.603,A -85,B 0,C 180,E1 -5556.436,E2 -5556.436} C_VEL
LIN {X 0,Y 509.92,Z 320.592,A -85,B 0,C 180,E1 -5559.845,E2 -5559.845} C_VEL
LIN {X 0,Y 509.871,Z 320.592,A -85,B 0,C 180,E1 -5563.174,E2 -5563.174} C_VEL
LIN {X 0,Y 509.865,Z 320.597,A -85,B 0,C 180,E1 -5565.634,E2 -5565.634} C_VEL
LIN {X 0,Y 509.915,Z 320.588,A -85,B 0,C 180,E1 -5568.875,E2 -5568.875} C_VEL
LIN {X 0,Y 509.888,Z 320.596,A -85,B 0,C 180,E1 -5572.078,E2 -5572.078} C_VEL
LIN {X 0,Y 509.967,Z 320.584,A -85,B 0,C 180,E1 -5574.464,E2 -5574.464} C_VEL
LIN {X 0,Y 510.047,Z 320.573,A -85,B 0,C 180,E1 -5577.631,E2 -5577.631} C_VEL
LIN {X 0,Y 510.038,Z 320.579,A -85,B 0,C 180,E1 -5580,E2 -5580} C_VEL
LIN {X 0,Y 510.051,Z 320.572,A -85,B 0,C 180,E1 -5582.369,E2 -5582.369} C_VEL
LIN {X 0,Y 509.941,Z 320.59,A -85,B 0,C 180,E1 -5585.536,E2 -5585.536} C_VEL
LIN {X 0,Y 509.892,Z 320.591,A -85,B 0,C 180,E1 -5588.721,E2 -5588.721} C_VEL
LIN {X 0,Y 509.909,Z 320.594,A -85,B 0,C 180,E1 -5591.932,E2 -5591.932} C_VEL
LIN {X 0,Y 509.9,Z 320.593,A -85,B 0,C 180,E1 -5595.242,E2 -5595.242} C_VEL
LIN {X 0,Y 509.836,Z 320.599,A -85,B 0,C 180,E1 -5598.485,E2 -5598.485} C_VEL
LIN {X 0,Y 509.822,Z 320.598,A -85,B 0,C 180,E1 -5601.003,E2 -5601.003} C_VEL
LIN {X 0,Y 509.812,Z 320.609,A -85,B 0,C 180,E1 -5603.565,E2 -5603.565} C_VEL
LIN {X 0,Y 509.819,Z 320.601,A -85,B 0,C 180,E1 -5606.356,E2 -5606.356} C_VEL
LIN {X 0,Y 509.797,Z 320.601,A -85,B 0,C 180,E1 -5608.85,E2 -5608.85} C_VEL
LIN {X 0,Y 509.792,Z 320.605,A -85,B 0,C 180,E1 -5611.593,E2 -5611.593} C_VEL
LIN {X 0,Y 509.836,Z 320.598,A -85,B 0,C 180,E1 -5614.415,E2 -5614.415} C_VEL
LIN {X 0,Y 509.774,Z 320.606,A -85,B 0,C 180,E1 -5617.345,E2 -5617.345} C_VEL
LIN {X 0,Y 509.789,Z 320.603,A -85,B 0,C 180,E1 -5620.387,E2 -5620.387} C_VEL
LIN {X 0,Y 509.794,Z 320.61,A -85,B 0,C 180,E1 -5623.575,E2 -5623.575} C_VEL
LIN {X 0,Y 509.794,Z 320.602,A -85,B 0,C 180,E1 -5626.425,E2 -5626.425} C_VEL
LIN {X 0,Y 509.788,Z 320.61,A -85,B 0,C 180,E1 -5629.613,E2 -5629.613} C_VEL
LIN {X 0,Y 509.762,Z 320.611,A -85,B 0,C 180,E1 -5632.654,E2 -5632.654} C_VEL
LIN {X 0,Y 509.758,Z 320.612,A -85,B 0,C 180,E1 -5633.692,E2 -5633.692} C_VEL
LIN {X 0,Y 509.097,Z 320.692,A -85,B 0,C 180,E1 -5634.352,E2 -5634.352} C_VEL
LIN {X 0,Y 506.279,Z 321.048,A -85,B 0,C 180,E1 -5635.425,E2 -5635.425} C_VEL
LIN {X 0,Y 503.89,Z 321.347,A -85,B 0,C 180,E1 -5636.288,E2 -5636.288} C_VEL
LIN {X 0,Y 502.851,Z 321.474,A -85,B 0,C 180,E1 -5636.955,E2 -5636.955} C_VEL
LIN {X 0,Y 502.76,Z 321.483,A -85,B 0,C 180,E1 -5637.181,E2 -5637.181} C_VEL
LIN {X 0,Y 502.747,Z 321.486,A -85,B 0,C 180,E1 -5640.079,E2 -5640.079} C_VEL
LIN {X 0,Y 502.804,Z 321.599,A -85,B 0,C 180,E1 -5641.779,E2 -5641.779} C_VEL
LIN {X 0,Y 504.555,Z 330.743,A -85,B 0,C 180,E1 -5643.53,E2 -5643.53} C_VEL
LIN {X 0,Y 504.121,Z 344.183,A -85,B 0,C 180,E1 -5645.899,E2 -5645.899} C_VEL
LIN {X 0,Y 507.011,Z 358.035,A -85,B 0,C 180,E1 -5646.222,E2 -5646.222} C_VEL
LIN {X 0,Y 506.199,Z 480.855,A -85,B 0,C 180,E1 -5648.01,E2 -5648.01} C_VEL
LIN {X 0,Y 505.866,Z 495.177,A -85,B 0,C 180,E1 -5648.379,E2 -5648.379} C_VEL
LIN {X 0,Y 505.481,Z 509.245,A -85,B 0,C 180,E1 -5648.915,E2 -5648.915} C_VEL
LIN {X 0,Y 505.075,Z 521.561,A -85,B 0,C 180,E1 -5649.536,E2 -5649.536} C_VEL
LIN {X 0,Y 504.618,Z 534.485,A -85,B 0,C 180,E1 -5650.367,E2 -5650.367} C_VEL
LIN {X 0,Y 504.151,Z 546.183,A -85,B 0,C 180,E1 -5651.299,E2 -5651.299} C_VEL
LIN {X 0,Y 503.65,Z 556.861,A -85,B 0,C 180,E1 -5652.332,E2 -5652.332} C_VEL
LIN {X 0,Y 503.22,Z 567.422,A -85,B 0,C 180,E1 -5653.572,E2 -5653.572} C_VEL
LIN {X 0,Y 502.848,Z 575.934,A -85,B 0,C 180,E1 -5654.785,E2 -5654.785} C_VEL
LIN {X 0,Y 502.549,Z 584.317,A -85,B 0,C 180,E1 -5656.247,E2 -5656.247} C_VEL
LIN {X 0,Y 502.382,Z 590.075,A -85,B 0,C 180,E1 -5657.477,E2 -5657.477} C_VEL
LIN {X 0,Y 502.209,Z 596.1,A -85,B 0,C 180,E1 -5659.11,E2 -5659.11} C_VEL
LIN {X 0,Y 502.106,Z 599.558,A -85,B 0,C 180,E1 -5660.33,E2 -5660.33} C_VEL
LIN {X 0,Y 502.097,Z 602.854,A -85,B 0,C 180,E1 -5661.954,E2 -5661.954} C_VEL
LIN {X 0,Y 502.091,Z 604.73,A -85,B 0,C 180,E1 -5663.57,E2 -5663.57} C_VEL
LIN {X 0,Y 502.046,Z 605.27,A -85,B 0,C 180,E1 -5665.182,E2 -5665.182} C_VEL
LIN {X 0,Y 502.101,Z 604.489,A -85,B 0,C 180,E1 -5666.79,E2 -5666.79} C_VEL
LIN {X 0,Y 502.039,Z 602.389,A -85,B 0,C 180,E1 -5668.396,E2 -5668.396} C_VEL
LIN {X 0,Y 502.04,Z 598.92,A -85,B 0,C 180,E1 -5670,E2 -5670} C_VEL
LIN {X 0,Y 502.228,Z 595.381,A -85,B 0,C 180,E1 -5671.203,E2 -5671.203} C_VEL
LIN {X 0,Y 502.446,Z 589.202,A -85,B 0,C 180,E1 -5672.806,E2 -5672.806} C_VEL
LIN {X 0,Y 502.642,Z 582.344,A -85,B 0,C 180,E1 -5674.21,E2 -5674.21} C_VEL
LIN {X 0,Y 503.003,Z 573.859,A -85,B 0,C 180,E1 -5675.613,E2 -5675.613} C_VEL
LIN {X 0,Y 503.375,Z 565.013,A -85,B 0,C 180,E1 -5676.816,E2 -5676.816} C_VEL
LIN {X 0,Y 503.71,Z 555.634,A -85,B 0,C 180,E1 -5677.884,E2 -5677.884} C_VEL
LIN {X 0,Y 504.192,Z 544.666,A -85,B 0,C 180,E1 -5678.921,E2 -5678.921} C_VEL
LIN {X 0,Y 504.666,Z 533.07,A -85,B 0,C 180,E1 -5679.822,E2 -5679.822} C_VEL
LIN {X 0,Y 505.153,Z 520.31,A -85,B 0,C 180,E1 -5680.623,E2 -5680.623} C_VEL
LIN {X 0,Y 505.54,Z 507.043,A -85,B 0,C 180,E1 -5681.274,E2 -5681.274} C_VEL
LIN {X 0,Y 505.921,Z 493.211,A -85,B 0,C 180,E1 -5681.773,E2 -5681.773} C_VEL
LIN {X 0,Y 506.176,Z 478.585,A -85,B 0,C 180,E1 -5682.123,E2 -5682.123} C_VEL
LIN {X 0,Y 506.923,Z 357.485,A -85,B 0,C 180,E1 -5683.879,E2 -5683.879} C_VEL
LIN {X 0,Y 504.151,Z 344.024,A -85,B 0,C 180,E1 -5684.208,E2 -5684.208} C_VEL
LIN {X 0,Y 504.521,Z 330.445,A -85,B 0,C 180,E1 -5686.593,E2 -5686.593} C_VEL
LIN {X 0,Y 502.808,Z 321.481,A -85,B 0,C 180,E1 -5688.326,E2 -5688.326} C_VEL
LIN {X 0,Y 502.768,Z 321.485,A -85,B 0,C 180,E1 -5691.312,E2 -5691.312} C_VEL
LIN {X 0,Y 502.756,Z 321.482,A -85,B 0,C 180,E1 -5693.916,E2 -5693.916} C_VEL
LIN {X 0,Y 502.759,Z 321.487,A -85,B 0,C 180,E1 -5696.572,E2 -5696.572} C_VEL
LIN {X 0,Y 502.754,Z 321.482,A -85,B 0,C 180,E1 -5699.292,E2 -5699.292} C_VEL
LIN {X 0,Y 502.758,Z 321.481,A -85,B 0,C 180,E1 -5702.087,E2 -5702.087} C_VEL
LIN {X 0,Y 502.769,Z 321.485,A -85,B 0,C 180,E1 -5704.968,E2 -5704.968} C_VEL
LIN {X 0,Y 502.749,Z 321.486,A -85,B 0,C 180,E1 -5708.479,E2 -5708.479} C_VEL
LIN {X 0,Y 502.753,Z 321.483,A -85,B 0,C 180,E1 -5711.073,E2 -5711.073} C_VEL
LIN {X 0,Y 502.781,Z 321.484,A -85,B 0,C 180,E1 -5714.529,E2 -5714.529} C_VEL
LIN {X 0,Y 502.736,Z 321.483,A -85,B 0,C 180,E1 -5717.854,E2 -5717.854} C_VEL
LIN {X 0,Y 502.768,Z 321.481,A -85,B 0,C 180,E1 -5721.02,E2 -5721.02} C_VEL
LIN {X 0,Y 502.754,Z 321.483,A -85,B 0,C 180,E1 -5724.173,E2 -5724.173} C_VEL
LIN {X 0,Y 502.802,Z 321.473,A -85,B 0,C 180,E1 -5726.999,E2 -5726.999} C_VEL
LIN {X 0,Y 502.751,Z 321.484,A -85,B 0,C 180,E1 -5730.078,E2 -5730.078} C_VEL
LIN {X 0,Y 502.774,Z 321.482,A -85,B 0,C 180,E1 -5732.529,E2 -5732.529} C_VEL
LIN {X 0,Y 502.774,Z 321.478,A -85,B 0,C 180,E1 -5735.313,E2 -5735.313} C_VEL
LIN {X 0,Y 502.777,Z 321.477,A -85,B 0,C 180,E1 -5737.826,E2 -5737.826} C_VEL
LIN {X 0,Y 502.807,Z 321.472,A -85,B 0,C 180,E1 -5740.399,E2 -5740.399} C_VEL
LIN {X 0,Y 502.752,Z 321.481,A -85,B 0,C 180,E1 -5742.928,E2 -5742.928} C_VEL
LIN {X 0,Y 502.83,Z 321.47,A -85,B 0,C 180,E1 -5745.428,E2 -5745.428} C_VEL
LIN {X 0,Y 502.88,Z 321.455,A -85,B 0,C 180,E1 -5748.717,E2 -5748.717} C_VEL
LIN {X 0,Y 502.875,Z 321.467,A -85,B 0,C 180,E1 -5751.966,E2 -5751.966} C_VEL
LIN {X 0,Y 502.902,Z 321.466,A -85,B 0,C 180,E1 -5754.386,E2 -5754.386} C_VEL
LIN {X 0,Y 503.02,Z 321.448,A -85,B 0,C 180,E1 -5757.598,E2 -5757.598} C_VEL
LIN {X 0,Y 502.994,Z 321.448,A -85,B 0,C 180,E1 -5760.8,E2 -5760.8} C_VEL
LIN {X 0,Y 503.014,Z 321.452,A -85,B 0,C 180,E1 -5762.402,E2 -5762.402} C_VEL
LIN {X 0,Y 502.92,Z 321.461,A -85,B 0,C 180,E1 -5765.613,E2 -5765.613} C_VEL
LIN {X 0,Y 502.864,Z 321.466,A -85,B 0,C 180,E1 -5768.843,E2 -5768.843} C_VEL
LIN {X 0,Y 502.849,Z 321.475,A -85,B 0,C 180,E1 -5772.101,E2 -5772.101} C_VEL
LIN {X 0,Y 502.852,Z 321.469,A -85,B 0,C 180,E1 -5775.399,E2 -5775.399} C_VEL
LIN {X 0,Y 502.826,Z 321.47,A -85,B 0,C 180,E1 -5778.752,E2 -5778.752} C_VEL
LIN {X 0,Y 502.787,Z 321.478,A -85,B 0,C 180,E1 -5781.311,E2 -5781.311} C_VEL
LIN {X 0,Y 502.778,Z 321.484,A -85,B 0,C 180,E1 -5783.914,E2 -5783.914} C_VEL
LIN {X 0,Y 502.845,Z 321.469,A -85,B 0,C 180,E1 -5786.567,E2 -5786.567} C_VEL
LIN {X 0,Y 502.818,Z 321.479,A -85,B 0,C 180,E1 -5789.935,E2 -5789.935} C_VEL
LIN {X 0,Y 502.834,Z 321.471,A -85,B 0,C 180,E1 -5793.031,E2 -5793.031} C_VEL
LIN {X 0,Y 502.776,Z 321.483,A -85,B 0,C 180,E1 -5795.951,E2 -5795.951} C_VEL
LIN {X 0,Y 502.803,Z 321.475,A -85,B 0,C 180,E1 -5798.976,E2 -5798.976} C_VEL
LIN {X 0,Y 502.797,Z 321.478,A -85,B 0,C 180,E1 -5802.139,E2 -5802.139} C_VEL
LIN {X 0,Y 502.788,Z 321.484,A -85,B 0,C 180,E1 -5805.47,E2 -5805.47} C_VEL
LIN {X 0,Y 502.821,Z 321.474,A -85,B 0,C 180,E1 -5808.934,E2 -5808.934} C_VEL
LIN {X 0,Y 502.795,Z 321.479,A -85,B 0,C 180,E1 -5812.046,E2 -5812.046} C_VEL
LIN {X 0,Y 502.809,Z 321.48,A -85,B 0,C 180,E1 -5815.035,E2 -5815.035} C_VEL
LIN {X 0,Y 502.785,Z 321.48,A -85,B 0,C 180,E1 -5817.915,E2 -5817.915} C_VEL
LIN {X 0,Y 502.826,Z 321.475,A -85,B 0,C 180,E1 -5820.712,E2 -5820.712} C_VEL
LIN {X 0,Y 502.864,Z 321.526,A -85,B 0,C 180,E1 -5823.388,E2 -5823.388} C_VEL
LIN {X 0,Y 505.319,Z 333.388,A -85,B 0,C 180,E1 -5825.339,E2 -5825.339} C_VEL
LIN {X 0,Y 504.777,Z 351.962,A -85,B 0,C 180,E1 -5828.134,E2 -5828.134} C_VEL
LIN {X 0,Y 504.182,Z 370.167,A -85,B 0,C 180,E1 -5830.836,E2 -5830.836} C_VEL
LIN {X 0,Y 506.882,Z 386.468,A -85,B 0,C 180,E1 -5831.189,E2 -5831.189} C_VEL
LIN {X 0,Y 506.026,Z 508.595,A -85,B 0,C 180,E1 -5832.964,E2 -5832.964} C_VEL
LIN {X 0,Y 505.724,Z 523.342,A -85,B 0,C 180,E1 -5833.351,E2 -5833.351} C_VEL
LIN {X 0,Y 505.344,Z 536.495,A -85,B 0,C 180,E1 -5833.85,E2 -5833.85} C_VEL
LIN {X 0,Y 504.912,Z 550.472,A -85,B 0,C 180,E1 -5834.561,E2 -5834.561} C_VEL
LIN {X 0,Y 504.386,Z 562.976,A -85,B 0,C 180,E1 -5835.371,E2 -5835.371} C_VEL
LIN {X 0,Y 503.883,Z 574.405,A -85,B 0,C 180,E1 -5836.284,E2 -5836.284} C_VEL
LIN {X 0,Y 503.48,Z 584.914,A -85,B 0,C 180,E1 -5837.3,E2 -5837.3} C_VEL
LIN {X 0,Y 503.086,Z 595.365,A -85,B 0,C 180,E1 -5838.517,E2 -5838.517} C_VEL
LIN {X 0,Y 502.72,Z 603.99,A -85,B 0,C 180,E1 -5839.732,E2 -5839.732} C_VEL
LIN {X 0,Y 502.48,Z 612.253,A -85,B 0,C 180,E1 -5841.15,E2 -5841.15} C_VEL
LIN {X 0,Y 502.293,Z 618.036,A -85,B 0,C 180,E1 -5842.361,E2 -5842.361} C_VEL
LIN {X 0,Y 502.234,Z 622.777,A -85,B 0,C 180,E1 -5843.572,E2 -5843.572} C_VEL
LIN {X 0,Y 502.167,Z 626.617,A -85,B 0,C 180,E1 -5844.781,E2 -5844.781} C_VEL
LIN {X 0,Y 502.112,Z 629.575,A -85,B 0,C 180,E1 -5845.987,E2 -5845.987} C_VEL
LIN {X 0,Y 502.089,Z 632.283,A -85,B 0,C 180,E1 -5847.593,E2 -5847.593} C_VEL
LIN {X 0,Y 501.988,Z 633.622,A -85,B 0,C 180,E1 -5849.198,E2 -5849.198} C_VEL
LIN {X 0,Y 501.988,Z 633.622,A -85,B 0,C 180,E1 -5850.802,E2 -5850.802} C_VEL
LIN {X 0,Y 502.089,Z 632.283,A -85,B 0,C 180,E1 -5852.407,E2 -5852.407} C_VEL
LIN {X 0,Y 502.112,Z 629.573,A -85,B 0,C 180,E1 -5854.013,E2 -5854.013} C_VEL
LIN {X 0,Y 502.201,Z 625.421,A -85,B 0,C 180,E1 -5855.622,E2 -5855.622} C_VEL
LIN {X 0,Y 502.252,Z 619.7,A -85,B 0,C 180,E1 -5857.235,E2 -5857.235} C_VEL
LIN {X 0,Y 502.438,Z 613.254,A -85,B 0,C 180,E1 -5858.648,E2 -5858.648} C_VEL
LIN {X 0,Y 502.683,Z 605.246,A -85,B 0,C 180,E1 -5860.065,E2 -5860.065} C_VEL
LIN {X 0,Y 503.025,Z 596.874,A -85,B 0,C 180,E1 -5861.28,E2 -5861.28} C_VEL
LIN {X 0,Y 503.415,Z 586.156,A -85,B 0,C 180,E1 -5862.569,E2 -5862.569} C_VEL
LIN {X 0,Y 503.854,Z 575.556,A -85,B 0,C 180,E1 -5863.614,E2 -5863.614} C_VEL
LIN {X 0,Y 504.327,Z 564.38,A -85,B 0,C 180,E1 -5864.527,E2 -5864.527} C_VEL
LIN {X 0,Y 504.799,Z 552.213,A -85,B 0,C 180,E1 -5865.339,E2 -5865.339} C_VEL
LIN {X 0,Y 505.304,Z 538.716,A -85,B 0,C 180,E1 -5866.047,E2 -5866.047} C_VEL
LIN {X 0,Y 505.671,Z 524.609,A -85,B 0,C 180,E1 -5866.606,E2 -5866.606} C_VEL
LIN {X 0,Y 506.013,Z 510.836,A -85,B 0,C 180,E1 -5866.984,E2 -5866.984} C_VEL
LIN {X 0,Y 506.204,Z 490.505,A -85,B 0,C 180,E1 -5867.316,E2 -5867.316} C_VEL
LIN {X 0,Y 506.905,Z 386.401,A -85,B 0,C 180,E1 -5868.81,E2 -5868.81} C_VEL
LIN {X 0,Y 504.172,Z 370.134,A -85,B 0,C 180,E1 -5869.165,E2 -5869.165} C_VEL
LIN {X 0,Y 504.897,Z 347.734,A -85,B 0,C 180,E1 -5872.507,E2 -5872.507} C_VEL
LIN {X 0,Y 505.382,Z 333.586,A -85,B 0,C 180,E1 -5874.657,E2 -5874.657} C_VEL
LIN {X 0,Y 502.851,Z 321.477,A -85,B 0,C 180,E1 -5876.693,E2 -5876.693} C_VEL
LIN {X 0,Y 502.826,Z 321.474,A -85,B 0,C 180,E1 -5879.288,E2 -5879.288} C_VEL
LIN {X 0,Y 502.785,Z 321.479,A -85,B 0,C 180,E1 -5882.085,E2 -5882.085} C_VEL
LIN {X 0,Y 502.801,Z 321.48,A -85,B 0,C 180,E1 -5884.966,E2 -5884.966} C_VEL
LIN {X 0,Y 502.795,Z 321.478,A -85,B 0,C 180,E1 -5887.954,E2 -5887.954} C_VEL
LIN {X 0,Y 502.821,Z 321.474,A -85,B 0,C 180,E1 -5891.066,E2 -5891.066} C_VEL
LIN {X 0,Y 502.788,Z 321.483,A -85,B 0,C 180,E1 -5894.53,E2 -5894.53} C_VEL
LIN {X 0,Y 502.797,Z 321.477,A -85,B 0,C 180,E1 -5897.861,E2 -5897.861} C_VEL
LIN {X 0,Y 502.803,Z 321.475,A -85,B 0,C 180,E1 -5901.024,E2 -5901.024} C_VEL
LIN {X 0,Y 502.774,Z 321.482,A -85,B 0,C 180,E1 -5904.17,E2 -5904.17} C_VEL
LIN {X 0,Y 502.835,Z 321.47,A -85,B 0,C 180,E1 -5906.994,E2 -5906.994} C_VEL
LIN {X 0,Y 502.818,Z 321.478,A -85,B 0,C 180,E1 -5910.065,E2 -5910.065} C_VEL
LIN {X 0,Y 502.847,Z 321.468,A -85,B 0,C 180,E1 -5913.444,E2 -5913.444} C_VEL
LIN {X 0,Y 502.778,Z 321.484,A -85,B 0,C 180,E1 -5916.086,E2 -5916.086} C_VEL
LIN {X 0,Y 502.787,Z 321.478,A -85,B 0,C 180,E1 -5918.689,E2 -5918.689} C_VEL
LIN {X 0,Y 502.826,Z 321.47,A -85,B 0,C 180,E1 -5921.248,E2 -5921.248} C_VEL
LIN {X 0,Y 502.853,Z 321.47,A -85,B 0,C 180,E1 -5924.601,E2 -5924.601} C_VEL
LIN {X 0,Y 502.881,Z 321.47,A -85,B 0,C 180,E1 -5928.039,E2 -5928.039} C_VEL
LIN {X 0,Y 502.864,Z 321.465,A -85,B 0,C 180,E1 -5931.157,E2 -5931.157} C_VEL
LIN {X 0,Y 502.92,Z 321.462,A -85,B 0,C 180,E1 -5934.387,E2 -5934.387} C_VEL
LIN {X 0,Y 503.014,Z 321.448,A -85,B 0,C 180,E1 -5937.598,E2 -5937.598} C_VEL
LIN {X 0,Y 503.007,Z 321.454,A -85,B 0,C 180,E1 -5940,E2 -5940} C_VEL
LIN {X 0,Y 503.02,Z 321.447,A -85,B 0,C 180,E1 -5942.402,E2 -5942.402} C_VEL
LIN {X 0,Y 502.897,Z 321.468,A -85,B 0,C 180,E1 -5945.614,E2 -5945.614} C_VEL
LIN {X 0,Y 502.856,Z 321.473,A -85,B 0,C 180,E1 -5948.034,E2 -5948.034} C_VEL
LIN {X 0,Y 502.88,Z 321.466,A -85,B 0,C 180,E1 -5951.283,E2 -5951.283} C_VEL
LIN {X 0,Y 502.83,Z 321.471,A -85,B 0,C 180,E1 -5954.572,E2 -5954.572} C_VEL
LIN {X 0,Y 502.798,Z 321.478,A -85,B 0,C 180,E1 -5958.104,E2 -5958.104} C_VEL
LIN {X 0,Y 502.763,Z 321.48,A -85,B 0,C 180,E1 -5961.312,E2 -5961.312} C_VEL
LIN {X 0,Y 502.764,Z 321.481,A -85,B 0,C 180,E1 -5963.916,E2 -5963.916} C_VEL
LIN {X 0,Y 502.787,Z 321.476,A -85,B 0,C 180,E1 -5966.571,E2 -5966.571} C_VEL
LIN {X 0,Y 502.756,Z 321.481,A -85,B 0,C 180,E1 -5969.293,E2 -5969.293} C_VEL
LIN {X 0,Y 502.761,Z 321.48,A -85,B 0,C 180,E1 -5972.087,E2 -5972.087} C_VEL
LIN {X 0,Y 502.785,Z 321.479,A -85,B 0,C 180,E1 -5974.967,E2 -5974.967} C_VEL
LIN {X 0,Y 502.753,Z 321.48,A -85,B 0,C 180,E1 -5978.479,E2 -5978.479} C_VEL
LIN {X 0,Y 502.753,Z 321.484,A -85,B 0,C 180,E1 -5981.073,E2 -5981.073} C_VEL
LIN {X 0,Y 502.781,Z 321.478,A -85,B 0,C 180,E1 -5984.529,E2 -5984.529} C_VEL
LIN {X 0,Y 502.735,Z 321.486,A -85,B 0,C 180,E1 -5987.854,E2 -5987.854} C_VEL
LIN {X 0,Y 502.765,Z 321.486,A -85,B 0,C 180,E1 -5991.02,E2 -5991.02} C_VEL
LIN {X 0,Y 502.745,Z 321.483,A -85,B 0,C 180,E1 -5994.175,E2 -5994.175} C_VEL
LIN {X 0,Y 502.76,Z 321.483,A -85,B 0,C 180,E1 -5997.181,E2 -5997.181} C_VEL
LIN {X 0,Y 502.07,Z 321.568,A -85,B 0,C 180,E1 -5997.85,E2 -5997.85} C_VEL
LIN {X 0,Y 499.2,Z 321.93,A -85,B 0,C 180,E1 -5998.936,E2 -5998.936} C_VEL
LIN {X 0,Y 496.791,Z 322.229,A -85,B 0,C 180,E1 -5999.81,E2 -5999.81} C_VEL
LIN {X 0,Y 495.765,Z 322.357,A -85,B 0,C 180,E1 -6000.486,E2 -6000.486} C_VEL
LIN {X 0,Y 495.685,Z 322.365,A -85,B 0,C 180,E1 -6000.715,E2 -6000.715} C_VEL
LIN {X 0,Y 495.724,Z 322.373,A -85,B 0,C 180,E1 -6001.522,E2 -6001.522} C_VEL
LIN {X 0,Y 497.596,Z 331.778,A -85,B 0,C 180,E1 -6003.357,E2 -6003.357} C_VEL
LIN {X 0,Y 497.283,Z 344.332,A -85,B 0,C 180,E1 -6005.61,E2 -6005.61} C_VEL
LIN {X 0,Y 500.317,Z 359.68,A -85,B 0,C 180,E1 -6005.978,E2 -6005.978} C_VEL
LIN {X 0,Y 499.457,Z 480.544,A -85,B 0,C 180,E1 -6007.761,E2 -6007.761} C_VEL
LIN {X 0,Y 499.113,Z 495.013,A -85,B 0,C 180,E1 -6008.134,E2 -6008.134} C_VEL
LIN {X 0,Y 498.763,Z 507.858,A -85,B 0,C 180,E1 -6008.617,E2 -6008.617} C_VEL
LIN {X 0,Y 498.324,Z 520.515,A -85,B 0,C 180,E1 -6009.247,E2 -6009.247} C_VEL
LIN {X 0,Y 497.77,Z 533.67,A -85,B 0,C 180,E1 -6010.085,E2 -6010.085} C_VEL
LIN {X 0,Y 497.243,Z 545.547,A -85,B 0,C 180,E1 -6011.029,E2 -6011.029} C_VEL
LIN {X 0,Y 496.74,Z 556.37,A -85,B 0,C 180,E1 -6012.078,E2 -6012.078} C_VEL
LIN {X 0,Y 496.247,Z 567.046,A -85,B 0,C 180,E1 -6013.334,E2 -6013.334} C_VEL
LIN {X 0,Y 495.843,Z 576.321,A -85,B 0,C 180,E1 -6014.667,E2 -6014.667} C_VEL
LIN {X 0,Y 495.541,Z 584.163,A -85,B 0,C 180,E1 -6016.048,E2 -6016.048} C_VEL
LIN {X 0,Y 495.35,Z 589.96,A -85,B 0,C 180,E1 -6017.296,E2 -6017.296} C_VEL
LIN {X 0,Y 495.157,Z 594.693,A -85,B 0,C 180,E1 -6018.538,E2 -6018.538} C_VEL
LIN {X 0,Y 495.048,Z 599.574,A -85,B 0,C 180,E1 -6020.191,E2 -6020.191} C_VEL
LIN {X 0,Y 495.004,Z 602.936,A -85,B 0,C 180,E1 -6021.838,E2 -6021.838} C_VEL
LIN {X 0,Y 495.016,Z 604.885,A -85,B 0,C 180,E1 -6023.478,E2 -6023.478} C_VEL
LIN {X 0,Y 494.968,Z 605.485,A -85,B 0,C 180,E1 -6025.113,E2 -6025.113} C_VEL
LIN {X 0,Y 495.021,Z 604.759,A -85,B 0,C 180,E1 -6026.744,E2 -6026.744} C_VEL
LIN {X 0,Y 494.966,Z 602.714,A -85,B 0,C 180,E1 -6028.373,E2 -6028.373} C_VEL
LIN {X 0,Y 494.954,Z 599.304,A -85,B 0,C 180,E1 -6030,E2 -6030} C_VEL
LIN {X 0,Y 495.156,Z 595.818,A -85,B 0,C 180,E1 -6031.22,E2 -6031.22} C_VEL
LIN {X 0,Y 495.394,Z 589.714,A -85,B 0,C 180,E1 -6032.846,E2 -6032.846} C_VEL
LIN {X 0,Y 495.604,Z 582.928,A -85,B 0,C 180,E1 -6034.27,E2 -6034.27} C_VEL
LIN {X 0,Y 495.985,Z 574.524,A -85,B 0,C 180,E1 -6035.692,E2 -6035.692} C_VEL
LIN {X 0,Y 496.383,Z 565.771,A -85,B 0,C 180,E1 -6036.912,E2 -6036.912} C_VEL
LIN {X 0,Y 496.7,Z 557.226,A -85,B 0,C 180,E1 -6037.919,E2 -6037.919} C_VEL
LIN {X 0,Y 497.217,Z 546.823,A -85,B 0,C 180,E1 -6038.945,E2 -6038.945} C_VEL
LIN {X 0,Y 497.683,Z 535.65,A -85,B 0,C 180,E1 -6039.859,E2 -6039.859} C_VEL
LIN {X 0,Y 498.176,Z 523.459,A -85,B 0,C 180,E1 -6040.671,E2 -6040.671} C_VEL
LIN {X 0,Y 498.662,Z 509.889,A -85,B 0,C 180,E1 -6041.38,E2 -6041.38} C_VEL
LIN {X 0,Y 499.1,Z 495.55,A -85,B 0,C 180,E1 -6041.936,E2 -6041.936} C_VEL
LIN {X 0,Y 499.364,Z 481.187,A -85,B 0,C 180,E1 -6042.316,E2 -6042.316} C_VEL
LIN {X 0,Y 500.22,Z 358.544,A -85,B 0,C 180,E1 -6044.126,E2 -6044.126} C_VEL
LIN {X 0,Y 497.237,Z 344.349,A -85,B 0,C 180,E1 -6044.456,E2 -6044.456} C_VEL
LIN {X 0,Y 497.618,Z 332.157,A -85,B 0,C 180,E1 -6046.618,E2 -6046.618} C_VEL
LIN {X 0,Y 495.75,Z 322.361,A -85,B 0,C 180,E1 -6048.51,E2 -6048.51} C_VEL
LIN {X 0,Y 495.733,Z 322.359,A -85,B 0,C 180,E1 -6051.63,E2 -6051.63} C_VEL
LIN {X 0,Y 495.704,Z 322.362,A -85,B 0,C 180,E1 -6054.278,E2 -6054.278} C_VEL
LIN {X 0,Y 495.72,Z 322.366,A -85,B 0,C 180,E1 -6056.98,E2 -6056.98} C_VEL
LIN {X 0,Y 495.697,Z 322.359,A -85,B 0,C 180,E1 -6059.751,E2 -6059.751} C_VEL
LIN {X 0,Y 495.726,Z 322.362,A -85,B 0,C 180,E1 -6062.598,E2 -6062.598} C_VEL
LIN {X 0,Y 495.721,Z 322.357,A -85,B 0,C 180,E1 -6065.54,E2 -6065.54} C_VEL
LIN {X 0,Y 495.727,Z 322.362,A -85,B 0,C 180,E1 -6068.762,E2 -6068.762} C_VEL
LIN {X 0,Y 495.703,Z 322.358,A -85,B 0,C 180,E1 -6071.787,E2 -6071.787} C_VEL
LIN {X 0,Y 495.734,Z 322.356,A -85,B 0,C 180,E1 -6075.142,E2 -6075.142} C_VEL
LIN {X 0,Y 495.703,Z 322.362,A -85,B 0,C 180,E1 -6078.213,E2 -6078.213} C_VEL
LIN {X 0,Y 495.713,Z 322.357,A -85,B 0,C 180,E1 -6081.404,E2 -6081.404} C_VEL
LIN {X 0,Y 495.731,Z 322.362,A -85,B 0,C 180,E1 -6084.46,E2 -6084.46} C_VEL
LIN {X 0,Y 495.744,Z 322.35,A -85,B 0,C 180,E1 -6087.403,E2 -6087.403} C_VEL
LIN {X 0,Y 495.703,Z 322.364,A -85,B 0,C 180,E1 -6090.249,E2 -6090.249} C_VEL
LIN {X 0,Y 495.742,Z 322.352,A -85,B 0,C 180,E1 -6093.271,E2 -6093.271} C_VEL
LIN {X 0,Y 495.713,Z 322.358,A -85,B 0,C 180,E1 -6095.723,E2 -6095.723} C_VEL
LIN {X 0,Y 495.736,Z 322.353,A -85,B 0,C 180,E1 -6098.37,E2 -6098.37} C_VEL
LIN {X 0,Y 495.768,Z 322.347,A -85,B 0,C 180,E1 -6100.971,E2 -6100.971} C_VEL
LIN {X 0,Y 495.806,Z 322.35,A -85,B 0,C 180,E1 -6104.558,E2 -6104.558} C_VEL
LIN {X 0,Y 495.833,Z 322.342,A -85,B 0,C 180,E1 -6107.965,E2 -6107.965} C_VEL
LIN {X 0,Y 495.835,Z 322.338,A -85,B 0,C 180,E1 -6111.03,E2 -6111.03} C_VEL
LIN {X 0,Y 495.829,Z 322.343,A -85,B 0,C 180,E1 -6113.489,E2 -6113.489} C_VEL
LIN {X 0,Y 495.728,Z 322.36,A -85,B 0,C 180,E1 -6115.935,E2 -6115.935} C_VEL
LIN {X 0,Y 495.988,Z 322.324,A -85,B 0,C 180,E1 -6117.563,E2 -6117.563} C_VEL
LIN {X 0,Y 495.945,Z 322.326,A -85,B 0,C 180,E1 -6120.812,E2 -6120.812} C_VEL
LIN {X 0,Y 495.981,Z 322.328,A -85,B 0,C 180,E1 -6122.436,E2 -6122.436} C_VEL
LIN {X 0,Y 495.875,Z 322.34,A -85,B 0,C 180,E1 -6125.693,E2 -6125.693} C_VEL
LIN {X 0,Y 495.835,Z 322.341,A -85,B 0,C 180,E1 -6128.97,E2 -6128.97} C_VEL
LIN {X 0,Y 495.832,Z 322.35,A -85,B 0,C 180,E1 -6132.034,E2 -6132.034} C_VEL
LIN {X 0,Y 495.827,Z 322.345,A -85,B 0,C 180,E1 -6135.451,E2 -6135.451} C_VEL
LIN {X 0,Y 495.782,Z 322.348,A -85,B 0,C 180,E1 -6139.028,E2 -6139.028} C_VEL
LIN {X 0,Y 495.746,Z 322.359,A -85,B 0,C 180,E1 -6141.629,E2 -6141.629} C_VEL
LIN {X 0,Y 495.753,Z 322.352,A -85,B 0,C 180,E1 -6144.866,E2 -6144.866} C_VEL
LIN {X 0,Y 495.746,Z 322.36,A -85,B 0,C 180,E1 -6147.893,E2 -6147.893} C_VEL
LIN {X 0,Y 495.754,Z 322.353,A -85,B 0,C 180,E1 -6150.687,E2 -6150.687} C_VEL
LIN {X 0,Y 495.762,Z 322.358,A -85,B 0,C 180,E1 -6153.564,E2 -6153.564} C_VEL
LIN {X 0,Y 495.73,Z 322.357,A -85,B 0,C 180,E1 -6156.544,E2 -6156.544} C_VEL
LIN {X 0,Y 495.758,Z 322.361,A -85,B 0,C 180,E1 -6159.638,E2 -6159.638} C_VEL
LIN {X 0,Y 495.739,Z 322.355,A -85,B 0,C 180,E1 -6162.507,E2 -6162.507} C_VEL
LIN {X 0,Y 495.739,Z 322.358,A -85,B 0,C 180,E1 -6165.141,E2 -6165.141} C_VEL
LIN {X 0,Y 495.758,Z 322.353,A -85,B 0,C 180,E1 -6168.219,E2 -6168.219} C_VEL
LIN {X 0,Y 495.752,Z 322.362,A -85,B 0,C 180,E1 -6171.408,E2 -6171.408} C_VEL
LIN {X 0,Y 495.757,Z 322.355,A -85,B 0,C 180,E1 -6174.463,E2 -6174.463} C_VEL
LIN {X 0,Y 495.769,Z 322.359,A -85,B 0,C 180,E1 -6177.406,E2 -6177.406} C_VEL
LIN {X 0,Y 495.768,Z 322.353,A -85,B 0,C 180,E1 -6180.254,E2 -6180.254} C_VEL
LIN {X 0,Y 495.829,Z 322.504,A -85,B 0,C 180,E1 -6183.181,E2 -6183.181} C_VEL
LIN {X 0,Y 498.364,Z 334.548,A -85,B 0,C 180,E1 -6185.194,E2 -6185.194} C_VEL
LIN {X 0,Y 497.989,Z 347.425,A -85,B 0,C 180,E1 -6187.163,E2 -6187.163} C_VEL
LIN {X 0,Y 497.311,Z 365.956,A -85,B 0,C 180,E1 -6189.958,E2 -6189.958} C_VEL
LIN {X 0,Y 497.224,Z 370.002,A -85,B 0,C 180,E1 -6190.566,E2 -6190.566} C_VEL
LIN {X 0,Y 500.173,Z 387.696,A -85,B 0,C 180,E1 -6190.95,E2 -6190.95} C_VEL
LIN {X 0,Y 499.239,Z 508.385,A -85,B 0,C 180,E1 -6192.726,E2 -6192.726} C_VEL
LIN {X 0,Y 498.891,Z 523.245,A -85,B 0,C 180,E1 -6193.12,E2 -6193.12} C_VEL
LIN {X 0,Y 498.468,Z 537.421,A -85,B 0,C 180,E1 -6193.674,E2 -6193.674} C_VEL
LIN {X 0,Y 498.055,Z 550.267,A -85,B 0,C 180,E1 -6194.343,E2 -6194.343} C_VEL
LIN {X 0,Y 497.478,Z 562.772,A -85,B 0,C 180,E1 -6195.164,E2 -6195.164} C_VEL
LIN {X 0,Y 496.902,Z 575.378,A -85,B 0,C 180,E1 -6196.192,E2 -6196.192} C_VEL
LIN {X 0,Y 496.439,Z 585.975,A -85,B 0,C 180,E1 -6197.252,E2 -6197.252} C_VEL
LIN {X 0,Y 496,Z 596.69,A -85,B 0,C 180,E1 -6198.558,E2 -6198.558} C_VEL
LIN {X 0,Y 495.626,Z 605.06,A -85,B 0,C 180,E1 -6199.79,E2 -6199.79} C_VEL
LIN {X 0,Y 495.371,Z 613.065,A -85,B 0,C 180,E1 -6201.227,E2 -6201.227} C_VEL
LIN {X 0,Y 495.173,Z 619.511,A -85,B 0,C 180,E1 -6202.661,E2 -6202.661} C_VEL
LIN {X 0,Y 495.118,Z 623.57,A -85,B 0,C 180,E1 -6203.763,E2 -6203.763} C_VEL
LIN {X 0,Y 495.03,Z 627.486,A -85,B 0,C 180,E1 -6205.113,E2 -6205.113} C_VEL
LIN {X 0,Y 495.033,Z 630.903,A -85,B 0,C 180,E1 -6206.745,E2 -6206.745} C_VEL
LIN {X 0,Y 494.959,Z 632.921,A -85,B 0,C 180,E1 -6208.373,E2 -6208.373} C_VEL
LIN {X 0,Y 494.896,Z 633.588,A -85,B 0,C 180,E1 -6210,E2 -6210} C_VEL
LIN {X 0,Y 494.959,Z 632.919,A -85,B 0,C 180,E1 -6211.627,E2 -6211.627} C_VEL
LIN {X 0,Y 495.033,Z 630.901,A -85,B 0,C 180,E1 -6213.256,E2 -6213.256} C_VEL
LIN {X 0,Y 495.03,Z 627.48,A -85,B 0,C 180,E1 -6214.887,E2 -6214.887} C_VEL
LIN {X 0,Y 495.13,Z 622.679,A -85,B 0,C 180,E1 -6216.487,E2 -6216.487} C_VEL
LIN {X 0,Y 495.21,Z 617.817,A -85,B 0,C 180,E1 -6217.749,E2 -6217.749} C_VEL
LIN {X 0,Y 495.44,Z 610.94,A -85,B 0,C 180,E1 -6219.183,E2 -6219.183} C_VEL
LIN {X 0,Y 495.772,Z 602.405,A -85,B 0,C 180,E1 -6220.62,E2 -6220.62} C_VEL
LIN {X 0,Y 496.146,Z 592.807,A -85,B 0,C 180,E1 -6221.941,E2 -6221.941} C_VEL
LIN {X 0,Y 496.545,Z 582.719,A -85,B 0,C 180,E1 -6223.089,E2 -6223.089} C_VEL
LIN {X 0,Y 497.018,Z 571.813,A -85,B 0,C 180,E1 -6224.118,E2 -6224.118} C_VEL
LIN {X 0,Y 497.605,Z 559.881,A -85,B 0,C 180,E1 -6225.042,E2 -6225.042} C_VEL
LIN {X 0,Y 498.16,Z 546.677,A -85,B 0,C 180,E1 -6225.863,E2 -6225.863} C_VEL
LIN {X 0,Y 498.626,Z 532.771,A -85,B 0,C 180,E1 -6226.527,E2 -6226.527} C_VEL
LIN {X 0,Y 499.031,Z 518.623,A -85,B 0,C 180,E1 -6227.02,E2 -6227.02} C_VEL
LIN {X 0,Y 499.299,Z 504.074,A -85,B 0,C 180,E1 -6227.351,E2 -6227.351} C_VEL
LIN {X 0,Y 500.218,Z 387.747,A -85,B 0,C 180,E1 -6229.05,E2 -6229.05} C_VEL
LIN {X 0,Y 497.224,Z 369.962,A -85,B 0,C 180,E1 -6229.443,E2 -6229.443} C_VEL
LIN {X 0,Y 497.983,Z 349.036,A -85,B 0,C 180,E1 -6232.618,E2 -6232.618} C_VEL
LIN {X 0,Y 498.489,Z 334.913,A -85,B 0,C 180,E1 -6234.799,E2 -6234.799} C_VEL
LIN {X 0,Y 495.823,Z 322.352,A -85,B 0,C 180,E1 -6236.974,E2 -6236.974} C_VEL
LIN {X 0,Y 495.767,Z 322.355,A -85,B 0,C 180,E1 -6240.147,E2 -6240.147} C_VEL
LIN {X 0,Y 495.795,Z 322.349,A -85,B 0,C 180,E1 -6243.245,E2 -6243.245} C_VEL
LIN {X 0,Y 495.722,Z 322.361,A -85,B 0,C 180,E1 -6246.089,E2 -6246.089} C_VEL
LIN {X 0,Y 495.765,Z 322.354,A -85,B 0,C 180,E1 -6248.768,E2 -6248.768} C_VEL
LIN {X 0,Y 495.758,Z 322.352,A -85,B 0,C 180,E1 -6251.781,E2 -6251.781} C_VEL
LIN {X 0,Y 495.739,Z 322.354,A -85,B 0,C 180,E1 -6255.141,E2 -6255.141} C_VEL
LIN {X 0,Y 495.758,Z 322.357,A -85,B 0,C 180,E1 -6258.219,E2 -6258.219} C_VEL
LIN {X 0,Y 495.752,Z 322.352,A -85,B 0,C 180,E1 -6261.409,E2 -6261.409} C_VEL
LIN {X 0,Y 495.748,Z 322.36,A -85,B 0,C 180,E1 -6264.462,E2 -6264.462} C_VEL
LIN {X 0,Y 495.771,Z 322.349,A -85,B 0,C 180,E1 -6267.406,E2 -6267.406} C_VEL
LIN {X 0,Y 495.766,Z 322.356,A -85,B 0,C 180,E1 -6270.254,E2 -6270.254} C_VEL
LIN {X 0,Y 495.777,Z 322.348,A -85,B 0,C 180,E1 -6273.263,E2 -6273.263} C_VEL
LIN {X 0,Y 495.746,Z 322.355,A -85,B 0,C 180,E1 -6276.613,E2 -6276.613} C_VEL
LIN {X 0,Y 495.782,Z 322.348,A -85,B 0,C 180,E1 -6279.324,E2 -6279.324} C_VEL
LIN {X 0,Y 495.782,Z 322.352,A -85,B 0,C 180,E1 -6281.829,E2 -6281.829} C_VEL
LIN {X 0,Y 495.828,Z 322.346,A -85,B 0,C 180,E1 -6284.549,E2 -6284.549} C_VEL
LIN {X 0,Y 495.833,Z 322.346,A -85,B 0,C 180,E1 -6287.966,E2 -6287.966} C_VEL
LIN {X 0,Y 495.835,Z 322.34,A -85,B 0,C 180,E1 -6291.03,E2 -6291.03} C_VEL
LIN {X 0,Y 495.875,Z 322.341,A -85,B 0,C 180,E1 -6294.307,E2 -6294.307} C_VEL
LIN {X 0,Y 495.981,Z 322.323,A -85,B 0,C 180,E1 -6297.564,E2 -6297.564} C_VEL
LIN {X 0,Y 495.976,Z 322.33,A -85,B 0,C 180,E1 -6300,E2 -6300} C_VEL
LIN {X 0,Y 495.988,Z 322.323,A -85,B 0,C 180,E1 -6302.437,E2 -6302.437} C_VEL
LIN {X 0,Y 495.855,Z 322.346,A -85,B 0,C 180,E1 -6305.694,E2 -6305.694} C_VEL
LIN {X 0,Y 495.82,Z 322.348,A -85,B 0,C 180,E1 -6308.149,E2 -6308.149} C_VEL
LIN {X 0,Y 495.855,Z 322.343,A -85,B 0,C 180,E1 -6311.445,E2 -6311.445} C_VEL
LIN {X 0,Y 495.781,Z 322.349,A -85,B 0,C 180,E1 -6314.783,E2 -6314.783} C_VEL
LIN {X 0,Y 495.776,Z 322.351,A -85,B 0,C 180,E1 -6318.235,E2 -6318.235} C_VEL
LIN {X 0,Y 495.75,Z 322.35,A -85,B 0,C 180,E1 -6320.758,E2 -6320.758} C_VEL
LIN {X 0,Y 495.738,Z 322.36,A -85,B 0,C 180,E1 -6323.388,E2 -6323.388} C_VEL
LIN {X 0,Y 495.72,Z 322.359,A -85,B 0,C 180,E1 -6326.072,E2 -6326.072} C_VEL
LIN {X 0,Y 495.699,Z 322.357,A -85,B 0,C 180,E1 -6328.82,E2 -6328.82} C_VEL
LIN {X 0,Y 495.734,Z 322.358,A -85,B 0,C 180,E1 -6331.72,E2 -6331.72} C_VEL
LIN {X 0,Y 495.758,Z 322.352,A -85,B 0,C 180,E1 -6334.691,E2 -6334.691} C_VEL
LIN {X 0,Y 495.697,Z 322.362,A -85,B 0,C 180,E1 -6337.565,E2 -6337.565} C_VEL
LIN {X 0,Y 495.709,Z 322.358,A -85,B 0,C 180,E1 -6340.04,E2 -6340.04} C_VEL
LIN {X 0,Y 495.693,Z 322.363,A -85,B 0,C 180,E1 -6342.887,E2 -6342.887} C_VEL
LIN {X 0,Y 495.716,Z 322.357,A -85,B 0,C 180,E1 -6345.997,E2 -6345.997} C_VEL
LIN {X 0,Y 495.71,Z 322.363,A -85,B 0,C 180,E1 -6349.294,E2 -6349.294} C_VEL
LIN {X 0,Y 495.71,Z 322.366,A -85,B 0,C 180,E1 -6351.404,E2 -6351.404} C_VEL
LIN {X 0,Y 495.722,Z 322.359,A -85,B 0,C 180,E1 -6354.46,E2 -6354.46} C_VEL
LIN {X 0,Y 495.727,Z 322.362,A -85,B 0,C 180,E1 -6357.402,E2 -6357.402} C_VEL
LIN {X 0,Y 495.699,Z 322.364,A -85,B 0,C 180,E1 -6360.249,E2 -6360.249} C_VEL
LIN {X 0,Y 495.685,Z 322.365,A -85,B 0,C 180,E1 -6360.715,E2 -6360.715} C_VEL
LIN {X 0,Y 495.473,Z 322.833,A -85,B 0,C 180,E1 -6361.163,E2 -6361.163} C_VEL
LIN {X 0,Y 494.934,Z 324.035,A -85,B 0,C 180,E1 -6361.592,E2 -6361.592} C_VEL
LIN {X 0,Y 493.326,Z 327.774,A -85,B 0,C 180,E1 -6362.389,E2 -6362.389} C_VEL
LIN {X 0,Y 491.626,Z 332.407,A -85,B 0,C 180,E1 -6363.153,E2 -6363.153} C_VEL
LIN {X 0,Y 490.691,Z 336.889,A -85,B 0,C 180,E1 -6363.931,E2 -6363.931} C_VEL
LIN {X 0,Y 490.395,Z 344.564,A -85,B 0,C 180,E1 -6365.319,E2 -6365.319} C_VEL
LIN {X 0,Y 493.674,Z 360.804,A -85,B 0,C 180,E1 -6365.716,E2 -6365.716} C_VEL
LIN {X 0,Y 492.712,Z 480.959,A -85,B 0,C 180,E1 -6367.514,E2 -6367.514} C_VEL
LIN {X 0,Y 492.35,Z 495.408,A -85,B 0,C 180,E1 -6367.895,E2 -6367.895} C_VEL
LIN {X 0,Y 491.956,Z 508.462,A -85,B 0,C 180,E1 -6368.397,E2 -6368.397} C_VEL
LIN {X 0,Y 491.471,Z 521.329,A -85,B 0,C 180,E1 -6369.053,E2 -6369.053} C_VEL
LIN {X 0,Y 490.885,Z 534.354,A -85,B 0,C 180,E1 -6369.903,E2 -6369.903} C_VEL
LIN {X 0,Y 490.336,Z 545.97,A -85,B 0,C 180,E1 -6370.846,E2 -6370.846} C_VEL
LIN {X 0,Y 489.867,Z 555.891,A -85,B 0,C 180,E1 -6371.818,E2 -6371.818} C_VEL
LIN {X 0,Y 489.297,Z 566.675,A -85,B 0,C 180,E1 -6373.09,E2 -6373.09} C_VEL
LIN {X 0,Y 488.911,Z 575.711,A -85,B 0,C 180,E1 -6374.391,E2 -6374.391} C_VEL
LIN {X 0,Y 488.527,Z 583.99,A -85,B 0,C 180,E1 -6375.844,E2 -6375.844} C_VEL
LIN {X 0,Y 488.304,Z 589.844,A -85,B 0,C 180,E1 -6377.11,E2 -6377.11} C_VEL
LIN {X 0,Y 488.105,Z 594.645,A -85,B 0,C 180,E1 -6378.371,E2 -6378.371} C_VEL
LIN {X 0,Y 487.99,Z 599.589,A -85,B 0,C 180,E1 -6380.048,E2 -6380.048} C_VEL
LIN {X 0,Y 487.927,Z 603.011,A -85,B 0,C 180,E1 -6381.718,E2 -6381.718} C_VEL
LIN {X 0,Y 487.934,Z 605.025,A -85,B 0,C 180,E1 -6383.383,E2 -6383.383} C_VEL
LIN {X 0,Y 487.891,Z 605.692,A -85,B 0,C 180,E1 -6385.042,E2 -6385.042} C_VEL
LIN {X 0,Y 487.943,Z 605.028,A -85,B 0,C 180,E1 -6386.697,E2 -6386.697} C_VEL
LIN {X 0,Y 487.895,Z 603.04,A -85,B 0,C 180,E1 -6388.349,E2 -6388.349} C_VEL
LIN {X 0,Y 487.872,Z 599.688,A -85,B 0,C 180,E1 -6390,E2 -6390} C_VEL
LIN {X 0,Y 488.086,Z 596.238,A -85,B 0,C 180,E1 -6391.238,E2 -6391.238} C_VEL
LIN {X 0,Y 488.107,Z 591.874,A -85,B 0,C 180,E1 -6392.476,E2 -6392.476} C_VEL
LIN {X 0,Y 488.479,Z 586.554,A -85,B 0,C 180,E1 -6393.712,E2 -6393.712} C_VEL
LIN {X 0,Y 488.801,Z 578.961,A -85,B 0,C 180,E1 -6395.156,E2 -6395.156} C_VEL
LIN {X 0,Y 489.171,Z 571.059,A -85,B 0,C 180,E1 -6396.393,E2 -6396.393} C_VEL
LIN {X 0,Y 489.526,Z 561.791,A -85,B 0,C 180,E1 -6397.604,E2 -6397.604} C_VEL
LIN {X 0,Y 490.131,Z 551.025,A -85,B 0,C 180,E1 -6398.763,E2 -6398.763} C_VEL
LIN {X 0,Y 490.69,Z 539.392,A -85,B 0,C 180,E1 -6399.793,E2 -6399.793} C_VEL
LIN {X 0,Y 491.224,Z 526.461,A -85,B 0,C 180,E1 -6400.719,E2 -6400.719} C_VEL
LIN {X 0,Y 491.758,Z 513.719,A -85,B 0,C 180,E1 -6401.437,E2 -6401.437} C_VEL
LIN {X 0,Y 492.225,Z 500.67,A -85,B 0,C 180,E1 -6402.001,E2 -6402.001} C_VEL
LIN {X 0,Y 492.47,Z 486.559,A -85,B 0,C 180,E1 -6402.439,E2 -6402.439} C_VEL
LIN {X 0,Y 492.656,Z 471.702,A -85,B 0,C 180,E1 -6402.722,E2 -6402.722} C_VEL
LIN {X 0,Y 493.554,Z 359.9,A -85,B 0,C 180,E1 -6404.368,E2 -6404.368} C_VEL
LIN {X 0,Y 490.351,Z 344.492,A -85,B 0,C 180,E1 -6404.738,E2 -6404.738} C_VEL
LIN {X 0,Y 490.707,Z 333.857,A -85,B 0,C 180,E1 -6406.645,E2 -6406.645} C_VEL
LIN {X 0,Y 488.981,Z 324.597,A -85,B 0,C 180,E1 -6408.433,E2 -6408.433} C_VEL
LIN {X 0,Y 488.708,Z 323.238,A -85,B 0,C 180,E1 -6408.699,E2 -6408.699} C_VEL
LIN {X 0,Y 488.703,Z 323.239,A -85,B 0,C 180,E1 -6411.071,E2 -6411.071} C_VEL
LIN {X 0,Y 488.664,Z 323.238,A -85,B 0,C 180,E1 -6413.747,E2 -6413.747} C_VEL
LIN {X 0,Y 488.669,Z 323.241,A -85,B 0,C 180,E1 -6416.477,E2 -6416.477} C_VEL
LIN {X 0,Y 488.662,Z 323.238,A -85,B 0,C 180,E1 -6419.275,E2 -6419.275} C_VEL
LIN {X 0,Y 488.681,Z 323.236,A -85,B 0,C 180,E1 -6422.149,E2 -6422.149} C_VEL
LIN {X 0,Y 488.7,Z 323.235,A -85,B 0,C 180,E1 -6425.117,E2 -6425.117} C_VEL
LIN {X 0,Y 488.646,Z 323.24,A -85,B 0,C 180,E1 -6428.203,E2 -6428.203} C_VEL
LIN {X 0,Y 488.646,Z 323.237,A -85,B 0,C 180,E1 -6431.422,E2 -6431.422} C_VEL
LIN {X 0,Y 488.699,Z 323.236,A -85,B 0,C 180,E1 -6434.803,E2 -6434.803} C_VEL
LIN {X 0,Y 488.651,Z 323.237,A -85,B 0,C 180,E1 -6437.469,E2 -6437.469} C_VEL
LIN {X 0,Y 488.67,Z 323.241,A -85,B 0,C 180,E1 -6440.742,E2 -6440.742} C_VEL
LIN {X 0,Y 488.648,Z 323.237,A -85,B 0,C 180,E1 -6443.865,E2 -6443.865} C_VEL
LIN {X 0,Y 488.711,Z 323.234,A -85,B 0,C 180,E1 -6446.521,E2 -6446.521} C_VEL
LIN {X 0,Y 488.669,Z 323.236,A -85,B 0,C 180,E1 -6449.777,E2 -6449.777} C_VEL
LIN {X 0,Y 488.684,Z 323.236,A -85,B 0,C 180,E1 -6452.599,E2 -6452.599} C_VEL
LIN {X 0,Y 488.698,Z 323.231,A -85,B 0,C 180,E1 -6455.351,E2 -6455.351} C_VEL
LIN {X 0,Y 488.691,Z 323.234,A -85,B 0,C 180,E1 -6458.042,E2 -6458.042} C_VEL
LIN {X 0,Y 488.73,Z 323.226,A -85,B 0,C 180,E1 -6460.686,E2 -6460.686} C_VEL
LIN {X 0,Y 488.674,Z 323.234,A -85,B 0,C 180,E1 -6463.283,E2 -6463.283} C_VEL
LIN {X 0,Y 488.726,Z 323.23,A -85,B 0,C 180,E1 -6465.85,E2 -6465.85} C_VEL
LIN {X 0,Y 488.809,Z 323.21,A -85,B 0,C 180,E1 -6468.387,E2 -6468.387} C_VEL
LIN {X 0,Y 488.783,Z 323.219,A -85,B 0,C 180,E1 -6471.733,E2 -6471.733} C_VEL
LIN {X 0,Y 488.82,Z 323.223,A -85,B 0,C 180,E1 -6474.224,E2 -6474.224} C_VEL
LIN {X 0,Y 488.955,Z 323.199,A -85,B 0,C 180,E1 -6477.528,E2 -6477.528} C_VEL
LIN {X 0,Y 488.898,Z 323.204,A -85,B 0,C 180,E1 -6480.823,E2 -6480.823} C_VEL
LIN {X 0,Y 488.947,Z 323.203,A -85,B 0,C 180,E1 -6482.471,E2 -6482.471} C_VEL
LIN {X 0,Y 488.832,Z 323.218,A -85,B 0,C 180,E1 -6485.776,E2 -6485.776} C_VEL
LIN {X 0,Y 488.774,Z 323.226,A -85,B 0,C 180,E1 -6488.267,E2 -6488.267} C_VEL
LIN {X 0,Y 488.809,Z 323.22,A -85,B 0,C 180,E1 -6491.612,E2 -6491.612} C_VEL
LIN {X 0,Y 488.765,Z 323.222,A -85,B 0,C 180,E1 -6495,E2 -6495} C_VEL
LIN {X 0,Y 488.749,Z 323.225,A -85,B 0,C 180,E1 -6498.442,E2 -6498.442} C_VEL
LIN {X 0,Y 488.71,Z 323.23,A -85,B 0,C 180,E1 -6501.07,E2 -6501.07} C_VEL
LIN {X 0,Y 488.68,Z 323.241,A -85,B 0,C 180,E1 -6503.746,E2 -6503.746} C_VEL
LIN {X 0,Y 488.728,Z 323.229,A -85,B 0,C 180,E1 -6506.473,E2 -6506.473} C_VEL
LIN {X 0,Y 488.713,Z 323.232,A -85,B 0,C 180,E1 -6509.271,E2 -6509.271} C_VEL
LIN {X 0,Y 488.706,Z 323.233,A -85,B 0,C 180,E1 -6512.147,E2 -6512.147} C_VEL
LIN {X 0,Y 488.72,Z 323.232,A -85,B 0,C 180,E1 -6515.115,E2 -6515.115} C_VEL
LIN {X 0,Y 488.681,Z 323.235,A -85,B 0,C 180,E1 -6518.2,E2 -6518.2} C_VEL
LIN {X 0,Y 488.72,Z 323.23,A -85,B 0,C 180,E1 -6520.344,E2 -6520.344} C_VEL
LIN {X 0,Y 488.686,Z 323.241,A -85,B 0,C 180,E1 -6523.654,E2 -6523.654} C_VEL
LIN {X 0,Y 488.686,Z 323.233,A -85,B 0,C 180,E1 -6526.345,E2 -6526.345} C_VEL
LIN {X 0,Y 488.735,Z 323.234,A -85,B 0,C 180,E1 -6529.676,E2 -6529.676} C_VEL
LIN {X 0,Y 488.683,Z 323.238,A -85,B 0,C 180,E1 -6532.841,E2 -6532.841} C_VEL
LIN {X 0,Y 488.736,Z 323.233,A -85,B 0,C 180,E1 -6535.887,E2 -6535.887} C_VEL
LIN {X 0,Y 488.694,Z 323.236,A -85,B 0,C 180,E1 -6538.82,E2 -6538.82} C_VEL
LIN {X 0,Y 488.746,Z 323.232,A -85,B 0,C 180,E1 -6541.671,E2 -6541.671} C_VEL
LIN {X 0,Y 488.793,Z 323.297,A -85,B 0,C 180,E1 -6542.942,E2 -6542.942} C_VEL
LIN {X 0,Y 491.409,Z 335.69,A -85,B 0,C 180,E1 -6545.045,E2 -6545.045} C_VEL
LIN {X 0,Y 491.272,Z 344.288,A -85,B 0,C 180,E1 -6546.387,E2 -6546.387} C_VEL
LIN {X 0,Y 490.582,Z 361.422,A -85,B 0,C 180,E1 -6549.013,E2 -6549.013} C_VEL
LIN {X 0,Y 490.291,Z 369.833,A -85,B 0,C 180,E1 -6550.294,E2 -6550.294} C_VEL
LIN {X 0,Y 493.437,Z 388.343,A -85,B 0,C 180,E1 -6550.699,E2 -6550.699} C_VEL
LIN {X 0,Y 492.456,Z 508.023,A -85,B 0,C 180,E1 -6552.48,E2 -6552.48} C_VEL
LIN {X 0,Y 492.106,Z 522.709,A -85,B 0,C 180,E1 -6552.872,E2 -6552.872} C_VEL
LIN {X 0,Y 491.654,Z 536.87,A -85,B 0,C 180,E1 -6553.427,E2 -6553.427} C_VEL
LIN {X 0,Y 491.201,Z 550.043,A -85,B 0,C 180,E1 -6554.119,E2 -6554.119} C_VEL
LIN {X 0,Y 490.556,Z 562.556,A -85,B 0,C 180,E1 -6554.949,E2 -6554.949} C_VEL
LIN {X 0,Y 489.964,Z 575.172,A -85,B 0,C 180,E1 -6555.992,E2 -6555.992} C_VEL
LIN {X 0,Y 489.434,Z 586.41,A -85,B 0,C 180,E1 -6557.14,E2 -6557.14} C_VEL
LIN {X 0,Y 488.971,Z 596.486,A -85,B 0,C 180,E1 -6558.391,E2 -6558.391} C_VEL
LIN {X 0,Y 488.596,Z 604.857,A -85,B 0,C 180,E1 -6559.642,E2 -6559.642} C_VEL
LIN {X 0,Y 488.312,Z 612.862,A -85,B 0,C 180,E1 -6561.099,E2 -6561.099} C_VEL
LIN {X 0,Y 488.083,Z 619.309,A -85,B 0,C 180,E1 -6562.554,E2 -6562.554} C_VEL
LIN {X 0,Y 488.018,Z 623.765,A -85,B 0,C 180,E1 -6563.796,E2 -6563.796} C_VEL
LIN {X 0,Y 487.96,Z 627.286,A -85,B 0,C 180,E1 -6565.042,E2 -6565.042} C_VEL
LIN {X 0,Y 487.955,Z 630.702,A -85,B 0,C 180,E1 -6566.697,E2 -6566.697} C_VEL
LIN {X 0,Y 487.887,Z 632.72,A -85,B 0,C 180,E1 -6568.349,E2 -6568.349} C_VEL
LIN {X 0,Y 487.817,Z 633.387,A -85,B 0,C 180,E1 -6570,E2 -6570} C_VEL
LIN {X 0,Y 487.887,Z 632.718,A -85,B 0,C 180,E1 -6571.651,E2 -6571.651} C_VEL
LIN {X 0,Y 487.955,Z 630.699,A -85,B 0,C 180,E1 -6573.303,E2 -6573.303} C_VEL
LIN {X 0,Y 487.961,Z 627.278,A -85,B 0,C 180,E1 -6574.958,E2 -6574.958} C_VEL
LIN {X 0,Y 488.04,Z 622.357,A -85,B 0,C 180,E1 -6576.615,E2 -6576.615} C_VEL
LIN {X 0,Y 488.231,Z 615.791,A -85,B 0,C 180,E1 -6578.276,E2 -6578.276} C_VEL
LIN {X 0,Y 488.469,Z 608.488,A -85,B 0,C 180,E1 -6579.733,E2 -6579.733} C_VEL
LIN {X 0,Y 488.882,Z 599.446,A -85,B 0,C 180,E1 -6581.191,E2 -6581.191} C_VEL
LIN {X 0,Y 489.269,Z 589.959,A -85,B 0,C 180,E1 -6582.443,E2 -6582.443} C_VEL
LIN {X 0,Y 489.776,Z 579.466,A -85,B 0,C 180,E1 -6583.59,E2 -6583.59} C_VEL
LIN {X 0,Y 490.289,Z 567.893,A -85,B 0,C 180,E1 -6584.634,E2 -6584.634} C_VEL
LIN {X 0,Y 490.938,Z 555.069,A -85,B 0,C 180,E1 -6585.57,E2 -6585.57} C_VEL
LIN {X 0,Y 491.436,Z 542.556,A -85,B 0,C 180,E1 -6586.3,E2 -6586.3} C_VEL
LIN {X 0,Y 491.918,Z 529.43,A -85,B 0,C 180,E1 -6586.892,E2 -6586.892} C_VEL
LIN {X 0,Y 492.3,Z 516.239,A -85,B 0,C 180,E1 -6587.327,E2 -6587.327} C_VEL
LIN {X 0,Y 492.6,Z 501.119,A -85,B 0,C 180,E1 -6587.649,E2 -6587.649} C_VEL
LIN {X 0,Y 493.433,Z 387.291,A -85,B 0,C 180,E1 -6589.334,E2 -6589.334} C_VEL
LIN {X 0,Y 490.338,Z 369.763,A -85,B 0,C 180,E1 -6589.737,E2 -6589.737} C_VEL
LIN {X 0,Y 491.145,Z 348.942,A -85,B 0,C 180,E1 -6592.95,E2 -6592.95} C_VEL
LIN {X 0,Y 491.684,Z 337.664,A -85,B 0,C 180,E1 -6594.714,E2 -6594.714} C_VEL
LIN {X 0,Y 490.08,Z 329.199,A -85,B 0,C 180,E1 -6596.166,E2 -6596.166} C_VEL
LIN {X 0,Y 488.775,Z 323.228,A -85,B 0,C 180,E1 -6597.262,E2 -6597.262} C_VEL
LIN {X 0,Y 488.712,Z 323.233,A -85,B 0,C 180,E1 -6600.363,E2 -6600.363} C_VEL
LIN {X 0,Y 488.736,Z 323.227,A -85,B 0,C 180,E1 -6603.484,E2 -6603.484} C_VEL
LIN {X 0,Y 488.684,Z 323.24,A -85,B 0,C 180,E1 -6606.355,E2 -6606.355} C_VEL
LIN {X 0,Y 488.703,Z 323.231,A -85,B 0,C 180,E1 -6609.254,E2 -6609.254} C_VEL
LIN {X 0,Y 488.709,Z 323.23,A -85,B 0,C 180,E1 -6611.6,E2 -6611.6} C_VEL
LIN {X 0,Y 488.703,Z 323.234,A -85,B 0,C 180,E1 -6614.803,E2 -6614.803} C_VEL
LIN {X 0,Y 488.694,Z 323.232,A -85,B 0,C 180,E1 -6617.475,E2 -6617.475} C_VEL
LIN {X 0,Y 488.735,Z 323.227,A -85,B 0,C 180,E1 -6619.677,E2 -6619.677} C_VEL
LIN {X 0,Y 488.673,Z 323.235,A -85,B 0,C 180,E1 -6622.841,E2 -6622.841} C_VEL
LIN {X 0,Y 488.733,Z 323.23,A -85,B 0,C 180,E1 -6625.887,E2 -6625.887} C_VEL
LIN {X 0,Y 488.695,Z 323.233,A -85,B 0,C 180,E1 -6628.821,E2 -6628.821} C_VEL
LIN {X 0,Y 488.715,Z 323.231,A -85,B 0,C 180,E1 -6631.669,E2 -6631.669} C_VEL
LIN {X 0,Y 488.716,Z 323.234,A -85,B 0,C 180,E1 -6634.443,E2 -6634.443} C_VEL
LIN {X 0,Y 488.725,Z 323.226,A -85,B 0,C 180,E1 -6637.153,E2 -6637.153} C_VEL
LIN {X 0,Y 488.728,Z 323.231,A -85,B 0,C 180,E1 -6639.811,E2 -6639.811} C_VEL
LIN {X 0,Y 488.714,Z 323.232,A -85,B 0,C 180,E1 -6642.423,E2 -6642.423} C_VEL
LIN {X 0,Y 488.765,Z 323.223,A -85,B 0,C 180,E1 -6645,E2 -6645} C_VEL
LIN {X 0,Y 488.809,Z 323.221,A -85,B 0,C 180,E1 -6648.388,E2 -6648.388} C_VEL
LIN {X 0,Y 488.774,Z 323.224,A -85,B 0,C 180,E1 -6651.733,E2 -6651.733} C_VEL
LIN {X 0,Y 488.832,Z 323.219,A -85,B 0,C 180,E1 -6654.224,E2 -6654.224} C_VEL
LIN {X 0,Y 488.947,Z 323.199,A -85,B 0,C 180,E1 -6657.529,E2 -6657.529} C_VEL
LIN {X 0,Y 488.945,Z 323.206,A -85,B 0,C 180,E1 -6660,E2 -6660} C_VEL
LIN {X 0,Y 488.955,Z 323.199,A -85,B 0,C 180,E1 -6662.472,E2 -6662.472} C_VEL
LIN {X 0,Y 488.815,Z 323.221,A -85,B 0,C 180,E1 -6665.776,E2 -6665.776} C_VEL
LIN {X 0,Y 488.768,Z 323.225,A -85,B 0,C 180,E1 -6668.268,E2 -6668.268} C_VEL
LIN {X 0,Y 488.81,Z 323.221,A -85,B 0,C 180,E1 -6671.613,E2 -6671.613} C_VEL
LIN {X 0,Y 488.751,Z 323.225,A -85,B 0,C 180,E1 -6675.001,E2 -6675.001} C_VEL
LIN {X 0,Y 488.718,Z 323.229,A -85,B 0,C 180,E1 -6678.444,E2 -6678.444} C_VEL
LIN {X 0,Y 488.694,Z 323.23,A -85,B 0,C 180,E1 -6681.072,E2 -6681.072} C_VEL
LIN {X 0,Y 488.669,Z 323.239,A -85,B 0,C 180,E1 -6683.747,E2 -6683.747} C_VEL
LIN {X 0,Y 488.685,Z 323.233,A -85,B 0,C 180,E1 -6686.477,E2 -6686.477} C_VEL
LIN {X 0,Y 488.663,Z 323.236,A -85,B 0,C 180,E1 -6689.275,E2 -6689.275} C_VEL
LIN {X 0,Y 488.688,Z 323.232,A -85,B 0,C 180,E1 -6692.149,E2 -6692.149} C_VEL
LIN {X 0,Y 488.709,Z 323.234,A -85,B 0,C 180,E1 -6695.116,E2 -6695.116} C_VEL
LIN {X 0,Y 488.65,Z 323.238,A -85,B 0,C 180,E1 -6698.203,E2 -6698.203} C_VEL
LIN {X 0,Y 488.647,Z 323.246,A -85,B 0,C 180,E1 -6701.422,E2 -6701.422} C_VEL
LIN {X 0,Y 488.699,Z 323.235,A -85,B 0,C 180,E1 -6704.804,E2 -6704.804} C_VEL
LIN {X 0,Y 488.651,Z 323.245,A -85,B 0,C 180,E1 -6707.47,E2 -6707.47} C_VEL
LIN {X 0,Y 488.668,Z 323.239,A -85,B 0,C 180,E1 -6710.742,E2 -6710.742} C_VEL
LIN {X 0,Y 488.64,Z 323.241,A -85,B 0,C 180,E1 -6713.864,E2 -6713.864} C_VEL
LIN {X 0,Y 488.695,Z 323.234,A -85,B 0,C 180,E1 -6716.524,E2 -6716.524} C_VEL
LIN {X 0,Y 488.655,Z 323.242,A -85,B 0,C 180,E1 -6719.649,E2 -6719.649} C_VEL
LIN {X 0,Y 488.708,Z 323.436,A -85,B 0,C 180,E1 -6721.311,E2 -6721.311} C_VEL
LIN {X 0,Y 490.632,Z 332.829,A -85,B 0,C 180,E1 -6723.178,E2 -6723.178} C_VEL
LIN {X 0,Y 490.691,Z 336.889,A -85,B 0,C 180,E1 -6723.931,E2 -6723.931} C_VEL
LIN {X 0,Y 489.979,Z 339.407,A -85,B 0,C 180,E1 -6724.305,E2 -6724.305} C_VEL
LIN {X 0,Y 488.542,Z 342.325,A -85,B 0,C 180,E1 -6724.613,E2 -6724.613} C_VEL
LIN {X 0,Y 486.482,Z 346.692,A -85,B 0,C 180,E1 -6724.937,E2 -6724.937} C_VEL
LIN {X 0,Y 485.398,Z 350.975,A -85,B 0,C 180,E1 -6725.15,E2 -6725.15} C_VEL
LIN {X 0,Y 485.573,Z 354.201,A -85,B 0,C 180,E1 -6725.258,E2 -6725.258} C_VEL
LIN {X 0,Y 487.023,Z 361.84,A -85,B 0,C 180,E1 -6725.441,E2 -6725.441} C_VEL
LIN {X 0,Y 485.979,Z 480.605,A -85,B 0,C 180,E1 -6727.241,E2 -6727.241} C_VEL
LIN {X 0,Y 485.653,Z 494.986,A -85,B 0,C 180,E1 -6727.618,E2 -6727.618} C_VEL
LIN {X 0,Y 485.219,Z 507.855,A -85,B 0,C 180,E1 -6728.11,E2 -6728.11} C_VEL
LIN {X 0,Y 484.702,Z 520.438,A -85,B 0,C 180,E1 -6728.747,E2 -6728.747} C_VEL
LIN {X 0,Y 484.098,Z 533.662,A -85,B 0,C 180,E1 -6729.609,E2 -6729.609} C_VEL
LIN {X 0,Y 483.578,Z 544.398,A -85,B 0,C 180,E1 -6730.472,E2 -6730.472} C_VEL
LIN {X 0,Y 482.989,Z 555.466,A -85,B 0,C 180,E1 -6731.549,E2 -6731.549} C_VEL
LIN {X 0,Y 482.468,Z 564.697,A -85,B 0,C 180,E1 -6732.625,E2 -6732.625} C_VEL
LIN {X 0,Y 482.021,Z 573.916,A -85,B 0,C 180,E1 -6733.917,E2 -6733.917} C_VEL
LIN {X 0,Y 481.636,Z 581.563,A -85,B 0,C 180,E1 -6735.205,E2 -6735.205} C_VEL
LIN {X 0,Y 481.323,Z 587.912,A -85,B 0,C 180,E1 -6736.489,E2 -6736.489} C_VEL
LIN {X 0,Y 481.116,Z 593.101,A -85,B 0,C 180,E1 -6737.771,E2 -6737.771} C_VEL
LIN {X 0,Y 480.965,Z 597.303,A -85,B 0,C 180,E1 -6739.049,E2 -6739.049} C_VEL
LIN {X 0,Y 480.842,Z 601.529,A -85,B 0,C 180,E1 -6740.748,E2 -6740.748} C_VEL
LIN {X 0,Y 480.84,Z 604.293,A -85,B 0,C 180,E1 -6742.441,E2 -6742.441} C_VEL
LIN {X 0,Y 480.82,Z 605.687,A -85,B 0,C 180,E1 -6744.127,E2 -6744.127} C_VEL
LIN {X 0,Y 480.783,Z 605.754,A -85,B 0,C 180,E1 -6745.809,E2 -6745.809} C_VEL
LIN {X 0,Y 480.84,Z 604.494,A -85,B 0,C 180,E1 -6747.487,E2 -6747.487} C_VEL
LIN {X 0,Y 480.769,Z 601.894,A -85,B 0,C 180,E1 -6749.162,E2 -6749.162} C_VEL
LIN {X 0,Y 480.941,Z 599.012,A -85,B 0,C 180,E1 -6750.419,E2 -6750.419} C_VEL
LIN {X 0,Y 481.092,Z 593.903,A -85,B 0,C 180,E1 -6752.093,E2 -6752.093} C_VEL
LIN {X 0,Y 481.26,Z 588.953,A -85,B 0,C 180,E1 -6753.349,E2 -6753.349} C_VEL
LIN {X 0,Y 481.646,Z 581.883,A -85,B 0,C 180,E1 -6754.813,E2 -6754.813} C_VEL
LIN {X 0,Y 482.063,Z 573.168,A -85,B 0,C 180,E1 -6756.277,E2 -6756.277} C_VEL
LIN {X 0,Y 482.394,Z 564.067,A -85,B 0,C 180,E1 -6757.534,E2 -6757.534} C_VEL
LIN {X 0,Y 483.102,Z 553.987,A -85,B 0,C 180,E1 -6758.681,E2 -6758.681} C_VEL
LIN {X 0,Y 483.605,Z 542.942,A -85,B 0,C 180,E1 -6759.726,E2 -6759.726} C_VEL
LIN {X 0,Y 484.201,Z 530.747,A -85,B 0,C 180,E1 -6760.665,E2 -6760.665} C_VEL
LIN {X 0,Y 484.752,Z 519.04,A -85,B 0,C 180,E1 -6761.393,E2 -6761.393} C_VEL
LIN {X 0,Y 485.196,Z 506.307,A -85,B 0,C 180,E1 -6762.018,E2 -6762.018} C_VEL
LIN {X 0,Y 485.613,Z 491.809,A -85,B 0,C 180,E1 -6762.538,E2 -6762.538} C_VEL
LIN {X 0,Y 485.857,Z 478.821,A -85,B 0,C 180,E1 -6762.85,E2 -6762.85} C_VEL
LIN {X 0,Y 486.779,Z 360.512,A -85,B 0,C 180,E1 -6764.629,E2 -6764.629} C_VEL
LIN {X 0,Y 483.445,Z 344.66,A -85,B 0,C 180,E1 -6765.022,E2 -6765.022} C_VEL
LIN {X 0,Y 483.723,Z 334.38,A -85,B 0,C 180,E1 -6766.893,E2 -6766.893} C_VEL
LIN {X 0,Y 481.692,Z 324.113,A -85,B 0,C 180,E1 -6768.943,E2 -6768.943} C_VEL
LIN {X 0,Y 481.639,Z 324.117,A -85,B 0,C 180,E1 -6771.395,E2 -6771.395} C_VEL
LIN {X 0,Y 481.643,Z 324.113,A -85,B 0,C 180,E1 -6774.115,E2 -6774.115} C_VEL
LIN {X 0,Y 481.644,Z 324.117,A -85,B 0,C 180,E1 -6777.114,E2 -6777.114} C_VEL
LIN {X 0,Y 481.602,Z 324.115,A -85,B 0,C 180,E1 -6779.747,E2 -6779.747} C_VEL
LIN {X 0,Y 481.636,Z 324.118,A -85,B 0,C 180,E1 -6782.677,E2 -6782.677} C_VEL
LIN {X 0,Y 481.644,Z 324.114,A -85,B 0,C 180,E1 -6785.2,E2 -6785.2} C_VEL
LIN {X 0,Y 481.622,Z 324.114,A -85,B 0,C 180,E1 -6788.002,E2 -6788.002} C_VEL
LIN {X 0,Y 481.607,Z 324.118,A -85,B 0,C 180,E1 -6791.047,E2 -6791.047} C_VEL
LIN {X 0,Y 481.653,Z 324.115,A -85,B 0,C 180,E1 -6794.459,E2 -6794.459} C_VEL
LIN {X 0,Y 481.615,Z 324.119,A -85,B 0,C 180,E1 -6796.856,E2 -6796.856} C_VEL
LIN {X 0,Y 481.63,Z 324.113,A -85,B 0,C 180,E1 -6800.054,E2 -6800.054} C_VEL
LIN {X 0,Y 481.607,Z 324.114,A -85,B 0,C 180,E1 -6803.251,E2 -6803.251} C_VEL
LIN {X 0,Y 481.674,Z 324.112,A -85,B 0,C 180,E1 -6806.327,E2 -6806.327} C_VEL
LIN {X 0,Y 481.615,Z 324.114,A -85,B 0,C 180,E1 -6809.425,E2 -6809.425} C_VEL
LIN {X 0,Y 481.648,Z 324.112,A -85,B 0,C 180,E1 -6812.164,E2 -6812.164} C_VEL
LIN {X 0,Y 481.677,Z 324.108,A -85,B 0,C 180,E1 -6814.967,E2 -6814.967} C_VEL
LIN {X 0,Y 481.64,Z 324.109,A -85,B 0,C 180,E1 -6817.704,E2 -6817.704} C_VEL
LIN {X 0,Y 481.696,Z 324.099,A -85,B 0,C 180,E1 -6820.392,E2 -6820.392} C_VEL
LIN {X 0,Y 481.618,Z 324.113,A -85,B 0,C 180,E1 -6823.031,E2 -6823.031} C_VEL
LIN {X 0,Y 481.677,Z 324.106,A -85,B 0,C 180,E1 -6825.638,E2 -6825.638} C_VEL
LIN {X 0,Y 481.755,Z 324.09,A -85,B 0,C 180,E1 -6828.215,E2 -6828.215} C_VEL
LIN {X 0,Y 481.739,Z 324.095,A -85,B 0,C 180,E1 -6831.611,E2 -6831.611} C_VEL
LIN {X 0,Y 481.781,Z 324.101,A -85,B 0,C 180,E1 -6834.139,E2 -6834.139} C_VEL
LIN {X 0,Y 481.921,Z 324.075,A -85,B 0,C 180,E1 -6837.492,E2 -6837.492} C_VEL
LIN {X 0,Y 481.85,Z 324.082,A -85,B 0,C 180,E1 -6840.835,E2 -6840.835} C_VEL
LIN {X 0,Y 481.913,Z 324.079,A -85,B 0,C 180,E1 -6842.507,E2 -6842.507} C_VEL
LIN {X 0,Y 481.791,Z 324.096,A -85,B 0,C 180,E1 -6845.861,E2 -6845.861} C_VEL
LIN {X 0,Y 481.732,Z 324.102,A -85,B 0,C 180,E1 -6848.389,E2 -6848.389} C_VEL
LIN {X 0,Y 481.754,Z 324.101,A -85,B 0,C 180,E1 -6851.785,E2 -6851.785} C_VEL
LIN {X 0,Y 481.746,Z 324.097,A -85,B 0,C 180,E1 -6855.224,E2 -6855.224} C_VEL
LIN {X 0,Y 481.71,Z 324.101,A -85,B 0,C 180,E1 -6858.722,E2 -6858.722} C_VEL
LIN {X 0,Y 481.649,Z 324.112,A -85,B 0,C 180,E1 -6861.394,E2 -6861.394} C_VEL
LIN {X 0,Y 481.661,Z 324.112,A -85,B 0,C 180,E1 -6864.114,E2 -6864.114} C_VEL
LIN {X 0,Y 481.7,Z 324.105,A -85,B 0,C 180,E1 -6867.127,E2 -6867.127} C_VEL
LIN {X 0,Y 481.676,Z 324.113,A -85,B 0,C 180,E1 -6869.741,E2 -6869.741} C_VEL
LIN {X 0,Y 481.675,Z 324.106,A -85,B 0,C 180,E1 -6872.674,E2 -6872.674} C_VEL
LIN {X 0,Y 481.639,Z 324.118,A -85,B 0,C 180,E1 -6875.709,E2 -6875.709} C_VEL
LIN {X 0,Y 481.672,Z 324.107,A -85,B 0,C 180,E1 -6878.859,E2 -6878.859} C_VEL
LIN {X 0,Y 481.654,Z 324.114,A -85,B 0,C 180,E1 -6881.913,E2 -6881.913} C_VEL
LIN {X 0,Y 481.656,Z 324.109,A -85,B 0,C 180,E1 -6884.458,E2 -6884.458} C_VEL
LIN {X 0,Y 481.649,Z 324.114,A -85,B 0,C 180,E1 -6887.839,E2 -6887.839} C_VEL
LIN {X 0,Y 481.682,Z 324.108,A -85,B 0,C 180,E1 -6890.651,E2 -6890.651} C_VEL
LIN {X 0,Y 481.632,Z 324.121,A -85,B 0,C 180,E1 -6893.375,E2 -6893.375} C_VEL
LIN {X 0,Y 481.711,Z 324.106,A -85,B 0,C 180,E1 -6896.33,E2 -6896.33} C_VEL
LIN {X 0,Y 481.652,Z 324.117,A -85,B 0,C 180,E1 -6899.417,E2 -6899.417} C_VEL
LIN {X 0,Y 481.712,Z 324.107,A -85,B 0,C 180,E1 -6902.559,E2 -6902.559} C_VEL
LIN {X 0,Y 481.746,Z 324.161,A -85,B 0,C 180,E1 -6902.707,E2 -6902.707} C_VEL
LIN {X 0,Y 484.633,Z 338.262,A -85,B 0,C 180,E1 -6905.131,E2 -6905.131} C_VEL
LIN {X 0,Y 483.861,Z 357.954,A -85,B 0,C 180,E1 -6908.209,E2 -6908.209} C_VEL
LIN {X 0,Y 483.324,Z 369.618,A -85,B 0,C 180,E1 -6910.009,E2 -6910.009} C_VEL
LIN {X 0,Y 486.709,Z 389.335,A -85,B 0,C 180,E1 -6910.451,E2 -6910.451} C_VEL
LIN {X 0,Y 485.686,Z 507.442,A -85,B 0,C 180,E1 -6912.228,E2 -6912.228} C_VEL
LIN {X 0,Y 485.315,Z 522.212,A -85,B 0,C 180,E1 -6912.622,E2 -6912.622} C_VEL
LIN {X 0,Y 484.874,Z 535.675,A -85,B 0,C 180,E1 -6913.149,E2 -6913.149} C_VEL
LIN {X 0,Y 484.371,Z 548.114,A -85,B 0,C 180,E1 -6913.791,E2 -6913.791} C_VEL
LIN {X 0,Y 483.735,Z 560.845,A -85,B 0,C 180,E1 -6914.624,E2 -6914.624} C_VEL
LIN {X 0,Y 483.13,Z 572.563,A -85,B 0,C 180,E1 -6915.575,E2 -6915.575} C_VEL
LIN {X 0,Y 482.523,Z 584.27,A -85,B 0,C 180,E1 -6916.738,E2 -6916.738} C_VEL
LIN {X 0,Y 482.1,Z 594.095,A -85,B 0,C 180,E1 -6917.926,E2 -6917.926} C_VEL
LIN {X 0,Y 481.663,Z 603.377,A -85,B 0,C 180,E1 -6919.278,E2 -6919.278} C_VEL
LIN {X 0,Y 481.298,Z 611.644,A -85,B 0,C 180,E1 -6920.757,E2 -6920.757} C_VEL
LIN {X 0,Y 481.078,Z 617.43,A -85,B 0,C 180,E1 -6922.022,E2 -6922.022} C_VEL
LIN {X 0,Y 480.963,Z 623.015,A -85,B 0,C 180,E1 -6923.534,E2 -6923.534} C_VEL
LIN {X 0,Y 480.891,Z 627.085,A -85,B 0,C 180,E1 -6924.969,E2 -6924.969} C_VEL
LIN {X 0,Y 480.878,Z 630.501,A -85,B 0,C 180,E1 -6926.649,E2 -6926.649} C_VEL
LIN {X 0,Y 480.789,Z 632.519,A -85,B 0,C 180,E1 -6928.325,E2 -6928.325} C_VEL
LIN {X 0,Y 480.741,Z 633.186,A -85,B 0,C 180,E1 -6930,E2 -6930} C_VEL
LIN {X 0,Y 480.789,Z 632.516,A -85,B 0,C 180,E1 -6931.675,E2 -6931.675} C_VEL
LIN {X 0,Y 480.879,Z 630.497,A -85,B 0,C 180,E1 -6933.351,E2 -6933.351} C_VEL
LIN {X 0,Y 480.891,Z 627.075,A -85,B 0,C 180,E1 -6935.031,E2 -6935.031} C_VEL
LIN {X 0,Y 480.959,Z 622.152,A -85,B 0,C 180,E1 -6936.713,E2 -6936.713} C_VEL
LIN {X 0,Y 481.149,Z 615.587,A -85,B 0,C 180,E1 -6938.399,E2 -6938.399} C_VEL
LIN {X 0,Y 481.423,Z 608.286,A -85,B 0,C 180,E1 -6939.877,E2 -6939.877} C_VEL
LIN {X 0,Y 481.877,Z 599.254,A -85,B 0,C 180,E1 -6941.355,E2 -6941.355} C_VEL
LIN {X 0,Y 482.303,Z 589.782,A -85,B 0,C 180,E1 -6942.626,E2 -6942.626} C_VEL
LIN {X 0,Y 482.83,Z 579.306,A -85,B 0,C 180,E1 -6943.789,E2 -6943.789} C_VEL
LIN {X 0,Y 483.391,Z 567.764,A -85,B 0,C 180,E1 -6944.848,E2 -6944.848} C_VEL
LIN {X 0,Y 484.065,Z 554.972,A -85,B 0,C 180,E1 -6945.797,E2 -6945.797} C_VEL
LIN {X 0,Y 484.597,Z 542.945,A -85,B 0,C 180,E1 -6946.512,E2 -6946.512} C_VEL
LIN {X 0,Y 485.132,Z 529.442,A -85,B 0,C 180,E1 -6947.135,E2 -6947.135} C_VEL
LIN {X 0,Y 485.537,Z 516.361,A -85,B 0,C 180,E1 -6947.577,E2 -6947.577} C_VEL
LIN {X 0,Y 485.831,Z 502.969,A -85,B 0,C 180,E1 -6947.876,E2 -6947.876} C_VEL
LIN {X 0,Y 486.798,Z 388.503,A -85,B 0,C 180,E1 -6949.599,E2 -6949.599} C_VEL
LIN {X 0,Y 483.403,Z 369.507,A -85,B 0,C 180,E1 -6950.054,E2 -6950.054} C_VEL
LIN {X 0,Y 484.324,Z 348.865,A -85,B 0,C 180,E1 -6953.293,E2 -6953.293} C_VEL
LIN {X 0,Y 484.817,Z 339.012,A -85,B 0,C 180,E1 -6954.859,E2 -6954.859} C_VEL
LIN {X 0,Y 482.308,Z 326.627,A -85,B 0,C 180,E1 -6957.041,E2 -6957.041} C_VEL
LIN {X 0,Y 481.709,Z 324.108,A -85,B 0,C 180,E1 -6957.501,E2 -6957.501} C_VEL
LIN {X 0,Y 481.647,Z 324.111,A -85,B 0,C 180,E1 -6960.711,E2 -6960.711} C_VEL
LIN {X 0,Y 481.699,Z 324.104,A -85,B 0,C 180,E1 -6963.733,E2 -6963.733} C_VEL
LIN {X 0,Y 481.627,Z 324.119,A -85,B 0,C 180,E1 -6966.747,E2 -6966.747} C_VEL
LIN {X 0,Y 481.679,Z 324.107,A -85,B 0,C 180,E1 -6969.941,E2 -6969.941} C_VEL
LIN {X 0,Y 481.634,Z 324.111,A -85,B 0,C 180,E1 -6973.147,E2 -6973.147} C_VEL
LIN {X 0,Y 481.656,Z 324.108,A -85,B 0,C 180,E1 -6975.642,E2 -6975.642} C_VEL
LIN {X 0,Y 481.659,Z 324.11,A -85,B 0,C 180,E1 -6978.959,E2 -6978.959} C_VEL
LIN {X 0,Y 481.653,Z 324.112,A -85,B 0,C 180,E1 -6981.994,E2 -6981.994} C_VEL
LIN {X 0,Y 481.69,Z 324.105,A -85,B 0,C 180,E1 -6985.318,E2 -6985.318} C_VEL
LIN {X 0,Y 481.649,Z 324.118,A -85,B 0,C 180,E1 -6988.312,E2 -6988.312} C_VEL
LIN {X 0,Y 481.677,Z 324.106,A -85,B 0,C 180,E1 -6991.217,E2 -6991.217} C_VEL
LIN {X 0,Y 481.67,Z 324.11,A -85,B 0,C 180,E1 -6994.041,E2 -6994.041} C_VEL
LIN {X 0,Y 481.677,Z 324.105,A -85,B 0,C 180,E1 -6996.812,E2 -6996.812} C_VEL
LIN {X 0,Y 481.699,Z 324.104,A -85,B 0,C 180,E1 -6999.503,E2 -6999.503} C_VEL
LIN {X 0,Y 481.692,Z 324.107,A -85,B 0,C 180,E1 -7002.158,E2 -7002.158} C_VEL
LIN {X 0,Y 481.746,Z 324.098,A -85,B 0,C 180,E1 -7004.776,E2 -7004.776} C_VEL
LIN {X 0,Y 481.755,Z 324.103,A -85,B 0,C 180,E1 -7008.215,E2 -7008.215} C_VEL
LIN {X 0,Y 481.733,Z 324.1,A -85,B 0,C 180,E1 -7011.611,E2 -7011.611} C_VEL
LIN {X 0,Y 481.791,Z 324.098,A -85,B 0,C 180,E1 -7014.139,E2 -7014.139} C_VEL
LIN {X 0,Y 481.913,Z 324.075,A -85,B 0,C 180,E1 -7017.493,E2 -7017.493} C_VEL
LIN {X 0,Y 481.914,Z 324.081,A -85,B 0,C 180,E1 -7020,E2 -7020} C_VEL
LIN {X 0,Y 481.921,Z 324.075,A -85,B 0,C 180,E1 -7022.508,E2 -7022.508} C_VEL
LIN {X 0,Y 481.777,Z 324.096,A -85,B 0,C 180,E1 -7025.861,E2 -7025.861} C_VEL
LIN {X 0,Y 481.726,Z 324.101,A -85,B 0,C 180,E1 -7028.389,E2 -7028.389} C_VEL
LIN {X 0,Y 481.756,Z 324.099,A -85,B 0,C 180,E1 -7031.785,E2 -7031.785} C_VEL
LIN {X 0,Y 481.733,Z 324.101,A -85,B 0,C 180,E1 -7035.225,E2 -7035.225} C_VEL
LIN {X 0,Y 481.66,Z 324.108,A -85,B 0,C 180,E1 -7038.724,E2 -7038.724} C_VEL
LIN {X 0,Y 481.633,Z 324.113,A -85,B 0,C 180,E1 -7041.396,E2 -7041.396} C_VEL
LIN {X 0,Y 481.649,Z 324.109,A -85,B 0,C 180,E1 -7044.115,E2 -7044.115} C_VEL
LIN {X 0,Y 481.655,Z 324.112,A -85,B 0,C 180,E1 -7047.117,E2 -7047.117} C_VEL
LIN {X 0,Y 481.603,Z 324.107,A -85,B 0,C 180,E1 -7049.747,E2 -7049.747} C_VEL
LIN {X 0,Y 481.649,Z 324.109,A -85,B 0,C 180,E1 -7052.676,E2 -7052.676} C_VEL
LIN {X 0,Y 481.652,Z 324.113,A -85,B 0,C 180,E1 -7055.202,E2 -7055.202} C_VEL
LIN {X 0,Y 481.626,Z 324.114,A -85,B 0,C 180,E1 -7058.002,E2 -7058.002} C_VEL
LIN {X 0,Y 481.607,Z 324.118,A -85,B 0,C 180,E1 -7061.047,E2 -7061.047} C_VEL
LIN {X 0,Y 481.653,Z 324.11,A -85,B 0,C 180,E1 -7064.459,E2 -7064.459} C_VEL
LIN {X 0,Y 481.615,Z 324.115,A -85,B 0,C 180,E1 -7066.856,E2 -7066.856} C_VEL
LIN {X 0,Y 481.63,Z 324.115,A -85,B 0,C 180,E1 -7070.055,E2 -7070.055} C_VEL
LIN {X 0,Y 481.603,Z 324.124,A -85,B 0,C 180,E1 -7073.251,E2 -7073.251} C_VEL
LIN {X 0,Y 481.674,Z 324.108,A -85,B 0,C 180,E1 -7076.327,E2 -7076.327} C_VEL
LIN {X 0,Y 481.614,Z 324.119,A -85,B 0,C 180,E1 -7079.426,E2 -7079.426} C_VEL
LIN {X 0,Y 481.649,Z 324.132,A -85,B 0,C 180,E1 -7081.019,E2 -7081.019} C_VEL
LIN {X 0,Y 483.821,Z 335.142,A -85,B 0,C 180,E1 -7083.236,E2 -7083.236} C_VEL
LIN {X 0,Y 483.516,Z 344.76,A -85,B 0,C 180,E1 -7085.011,E2 -7085.011} C_VEL
LIN {X 0,Y 485.573,Z 354.201,A -85,B 0,C 180,E1 -7085.258,E2 -7085.258} C_VEL
LIN {X 0,Y 485.626,Z 358.067,A -85,B 0,C 180,E1 -7085.32,E2 -7085.32} C_VEL
LIN {X 0,Y 484.554,Z 361.916,A -85,B 0,C 180,E1 -7085.332,E2 -7085.332} C_VEL
LIN {X 0,Y 480.918,Z 370.8,A -85,B 0,C 180,E1 -7085.305,E2 -7085.305} C_VEL
LIN {X 0,Y 480.248,Z 374.814,A -85,B 0,C 180,E1 -7085.337,E2 -7085.337} C_VEL
LIN {X 0,Y 479.285,Z 481.774,A -85,B 0,C 180,E1 -7086.991,E2 -7086.991} C_VEL
LIN {X 0,Y 478.909,Z 495.746,A -85,B 0,C 180,E1 -7087.371,E2 -7087.371} C_VEL
LIN {X 0,Y 478.444,Z 508.54,A -85,B 0,C 180,E1 -7087.872,E2 -7087.872} C_VEL
LIN {X 0,Y 477.879,Z 521.396,A -85,B 0,C 180,E1 -7088.541,E2 -7088.541} C_VEL
LIN {X 0,Y 477.25,Z 534.468,A -85,B 0,C 180,E1 -7089.416,E2 -7089.416} C_VEL
LIN {X 0,Y 476.656,Z 545.907,A -85,B 0,C 180,E1 -7090.366,E2 -7090.366} C_VEL
LIN {X 0,Y 475.991,Z 557.05,A -85,B 0,C 180,E1 -7091.491,E2 -7091.491} C_VEL
LIN {X 0,Y 475.366,Z 567.691,A -85,B 0,C 180,E1 -7092.801,E2 -7092.801} C_VEL
LIN {X 0,Y 474.894,Z 576.639,A -85,B 0,C 180,E1 -7094.144,E2 -7094.144} C_VEL
LIN {X 0,Y 474.45,Z 584.768,A -85,B 0,C 180,E1 -7095.634,E2 -7095.634} C_VEL
LIN {X 0,Y 474.172,Z 591.425,A -85,B 0,C 180,E1 -7097.154,E2 -7097.154} C_VEL
LIN {X 0,Y 473.903,Z 597.303,A -85,B 0,C 180,E1 -7098.884,E2 -7098.884} C_VEL
LIN {X 0,Y 473.759,Z 601.584,A -85,B 0,C 180,E1 -7100.608,E2 -7100.608} C_VEL
LIN {X 0,Y 473.753,Z 604.402,A -85,B 0,C 180,E1 -7102.327,E2 -7102.327} C_VEL
LIN {X 0,Y 473.737,Z 605.849,A -85,B 0,C 180,E1 -7104.039,E2 -7104.039} C_VEL
LIN {X 0,Y 473.69,Z 605.969,A -85,B 0,C 180,E1 -7105.746,E2 -7105.746} C_VEL
LIN {X 0,Y 473.756,Z 604.77,A -85,B 0,C 180,E1 -7107.449,E2 -7107.449} C_VEL
LIN {X 0,Y 473.697,Z 602.237,A -85,B 0,C 180,E1 -7109.15,E2 -7109.15} C_VEL
LIN {X 0,Y 473.759,Z 598.286,A -85,B 0,C 180,E1 -7110.85,E2 -7110.85} C_VEL
LIN {X 0,Y 473.989,Z 592.805,A -85,B 0,C 180,E1 -7112.549,E2 -7112.549} C_VEL
LIN {X 0,Y 474.368,Z 587.612,A -85,B 0,C 180,E1 -7113.823,E2 -7113.823} C_VEL
LIN {X 0,Y 474.728,Z 580.153,A -85,B 0,C 180,E1 -7115.309,E2 -7115.309} C_VEL
LIN {X 0,Y 475.161,Z 572.398,A -85,B 0,C 180,E1 -7116.582,E2 -7116.582} C_VEL
LIN {X 0,Y 475.601,Z 562.471,A -85,B 0,C 180,E1 -7117.929,E2 -7117.929} C_VEL
LIN {X 0,Y 476.275,Z 551.679,A -85,B 0,C 180,E1 -7119.127,E2 -7119.127} C_VEL
LIN {X 0,Y 476.877,Z 540.081,A -85,B 0,C 180,E1 -7120.186,E2 -7120.186} C_VEL
LIN {X 0,Y 477.504,Z 527.185,A -85,B 0,C 180,E1 -7121.138,E2 -7121.138} C_VEL
LIN {X 0,Y 478.165,Z 513.481,A -85,B 0,C 180,E1 -7121.928,E2 -7121.928} C_VEL
LIN {X 0,Y 478.597,Z 500.172,A -85,B 0,C 180,E1 -7122.509,E2 -7122.509} C_VEL
LIN {X 0,Y 478.92,Z 486.639,A -85,B 0,C 180,E1 -7122.932,E2 -7122.932} C_VEL
LIN {X 0,Y 479.123,Z 471.582,A -85,B 0,C 180,E1 -7123.223,E2 -7123.223} C_VEL
LIN {X 0,Y 480.07,Z 361.49,A -85,B 0,C 180,E1 -7124.887,E2 -7124.887} C_VEL
LIN {X 0,Y 476.555,Z 344.922,A -85,B 0,C 180,E1 -7125.294,E2 -7125.294} C_VEL
LIN {X 0,Y 476.852,Z 336.636,A -85,B 0,C 180,E1 -7126.816,E2 -7126.816} C_VEL
LIN {X 0,Y 474.653,Z 324.99,A -85,B 0,C 180,E1 -7129.151,E2 -7129.151} C_VEL
LIN {X 0,Y 474.583,Z 324.994,A -85,B 0,C 180,E1 -7131.729,E2 -7131.729} C_VEL
LIN {X 0,Y 474.622,Z 324.991,A -85,B 0,C 180,E1 -7134.495,E2 -7134.495} C_VEL
LIN {X 0,Y 474.596,Z 324.993,A -85,B 0,C 180,E1 -7137.327,E2 -7137.327} C_VEL
LIN {X 0,Y 474.552,Z 324.994,A -85,B 0,C 180,E1 -7140.234,E2 -7140.234} C_VEL
LIN {X 0,Y 474.61,Z 324.99,A -85,B 0,C 180,E1 -7143.223,E2 -7143.223} C_VEL
LIN {X 0,Y 474.567,Z 324.995,A -85,B 0,C 180,E1 -7146.326,E2 -7146.326} C_VEL
LIN {X 0,Y 474.6,Z 324.987,A -85,B 0,C 180,E1 -7149.551,E2 -7149.551} C_VEL
LIN {X 0,Y 474.568,Z 324.997,A -85,B 0,C 180,E1 -7152.94,E2 -7152.94} C_VEL
LIN {X 0,Y 474.583,Z 324.989,A -85,B 0,C 180,E1 -7155.891,E2 -7155.891} C_VEL
LIN {X 0,Y 474.583,Z 324.992,A -85,B 0,C 180,E1 -7159.047,E2 -7159.047} C_VEL
LIN {X 0,Y 474.587,Z 324.989,A -85,B 0,C 180,E1 -7161.708,E2 -7161.708} C_VEL
LIN {X 0,Y 474.613,Z 324.992,A -85,B 0,C 180,E1 -7164.724,E2 -7164.724} C_VEL
LIN {X 0,Y 474.62,Z 324.982,A -85,B 0,C 180,E1 -7167.786,E2 -7167.786} C_VEL
LIN {X 0,Y 474.58,Z 324.991,A -85,B 0,C 180,E1 -7170.895,E2 -7170.895} C_VEL
LIN {X 0,Y 474.592,Z 324.986,A -85,B 0,C 180,E1 -7173.624,E2 -7173.624} C_VEL
LIN {X 0,Y 474.637,Z 324.985,A -85,B 0,C 180,E1 -7176.642,E2 -7176.642} C_VEL
LIN {X 0,Y 474.646,Z 324.974,A -85,B 0,C 180,E1 -7180.089,E2 -7180.089} C_VEL
LIN {X 0,Y 474.593,Z 324.99,A -85,B 0,C 180,E1 -7182.772,E2 -7182.772} C_VEL
LIN {X 0,Y 474.636,Z 324.983,A -85,B 0,C 180,E1 -7185.42,E2 -7185.42} C_VEL
LIN {X 0,Y 474.709,Z 324.97,A -85,B 0,C 180,E1 -7188.037,E2 -7188.037} C_VEL
LIN {X 0,Y 474.712,Z 324.969,A -85,B 0,C 180,E1 -7191.486,E2 -7191.486} C_VEL
LIN {X 0,Y 474.744,Z 324.976,A -85,B 0,C 180,E1 -7194.052,E2 -7194.052} C_VEL
LIN {X 0,Y 474.887,Z 324.951,A -85,B 0,C 180,E1 -7197.455,E2 -7197.455} C_VEL
LIN {X 0,Y 474.884,Z 324.959,A -85,B 0,C 180,E1 -7200,E2 -7200} C_VEL
LIN {X 0,Y 474.878,Z 324.955,A -85,B 0,C 180,E1 -7202.544,E2 -7202.544} C_VEL
LIN {X 0,Y 474.752,Z 324.973,A -85,B 0,C 180,E1 -7205.948,E2 -7205.948} C_VEL
LIN {X 0,Y 474.707,Z 324.975,A -85,B 0,C 180,E1 -7208.514,E2 -7208.514} C_VEL
LIN {X 0,Y 474.708,Z 324.982,A -85,B 0,C 180,E1 -7211.962,E2 -7211.962} C_VEL
LIN {X 0,Y 474.703,Z 324.976,A -85,B 0,C 180,E1 -7215.455,E2 -7215.455} C_VEL
LIN {X 0,Y 474.665,Z 324.978,A -85,B 0,C 180,E1 -7219.01,E2 -7219.01} C_VEL
LIN {X 0,Y 474.592,Z 324.995,A -85,B 0,C 180,E1 -7221.729,E2 -7221.729} C_VEL
LIN {X 0,Y 474.642,Z 324.983,A -85,B 0,C 180,E1 -7224.494,E2 -7224.494} C_VEL
LIN {X 0,Y 474.657,Z 324.984,A -85,B 0,C 180,E1 -7227.328,E2 -7227.328} C_VEL
LIN {X 0,Y 474.607,Z 324.988,A -85,B 0,C 180,E1 -7230.81,E2 -7230.81} C_VEL
LIN {X 0,Y 474.64,Z 324.988,A -85,B 0,C 180,E1 -7233.984,E2 -7233.984} C_VEL
LIN {X 0,Y 474.574,Z 324.993,A -85,B 0,C 180,E1 -7236.899,E2 -7236.899} C_VEL
LIN {X 0,Y 474.63,Z 324.993,A -85,B 0,C 180,E1 -7239.647,E2 -7239.647} C_VEL
LIN {X 0,Y 474.616,Z 324.988,A -85,B 0,C 180,E1 -7242.934,E2 -7242.934} C_VEL
LIN {X 0,Y 474.608,Z 324.991,A -85,B 0,C 180,E1 -7245.895,E2 -7245.895} C_VEL
LIN {X 0,Y 474.629,Z 324.988,A -85,B 0,C 180,E1 -7249.041,E2 -7249.041} C_VEL
LIN {X 0,Y 474.612,Z 324.995,A -85,B 0,C 180,E1 -7251.704,E2 -7251.704} C_VEL
LIN {X 0,Y 474.631,Z 324.989,A -85,B 0,C 180,E1 -7254.726,E2 -7254.726} C_VEL
LIN {X 0,Y 474.637,Z 324.988,A -85,B 0,C 180,E1 -7257.788,E2 -7257.788} C_VEL
LIN {X 0,Y 474.626,Z 324.99,A -85,B 0,C 180,E1 -7260.884,E2 -7260.884} C_VEL
LIN {X 0,Y 474.683,Z 325.014,A -85,B 0,C 180,E1 -7262.464,E2 -7262.464} C_VEL
LIN {X 0,Y 477.693,Z 339.38,A -85,B 0,C 180,E1 -7264.977,E2 -7264.977} C_VEL
LIN {X 0,Y 476.967,Z 357.842,A -85,B 0,C 180,E1 -7267.908,E2 -7267.908} C_VEL
LIN {X 0,Y 476.392,Z 369.446,A -85,B 0,C 180,E1 -7269.727,E2 -7269.727} C_VEL
LIN {X 0,Y 479.991,Z 390.286,A -85,B 0,C 180,E1 -7270.198,E2 -7270.198} C_VEL
LIN {X 0,Y 478.875,Z 507.873,A -85,B 0,C 180,E1 -7271.994,E2 -7271.994} C_VEL
LIN {X 0,Y 478.485,Z 522.575,A -85,B 0,C 180,E1 -7272.399,E2 -7272.399} C_VEL
LIN {X 0,Y 477.962,Z 537.075,A -85,B 0,C 180,E1 -7272.987,E2 -7272.987} C_VEL
LIN {X 0,Y 477.44,Z 549.524,A -85,B 0,C 180,E1 -7273.66,E2 -7273.66} C_VEL
LIN {X 0,Y 476.779,Z 561.938,A -85,B 0,C 180,E1 -7274.504,E2 -7274.504} C_VEL
LIN {X 0,Y 476.061,Z 574.614,A -85,B 0,C 180,E1 -7275.574,E2 -7275.574} C_VEL
LIN {X 0,Y 475.464,Z 585.91,A -85,B 0,C 180,E1 -7276.755,E2 -7276.755} C_VEL
LIN {X 0,Y 474.964,Z 596.02,A -85,B 0,C 180,E1 -7278.044,E2 -7278.044} C_VEL
LIN {X 0,Y 474.565,Z 604.415,A -85,B 0,C 180,E1 -7279.332,E2 -7279.332} C_VEL
LIN {X 0,Y 474.201,Z 612.436,A -85,B 0,C 180,E1 -7280.832,E2 -7280.832} C_VEL
LIN {X 0,Y 473.953,Z 618.893,A -85,B 0,C 180,E1 -7282.331,E2 -7282.331} C_VEL
LIN {X 0,Y 473.833,Z 624.616,A -85,B 0,C 180,E1 -7284.04,E2 -7284.04} C_VEL
LIN {X 0,Y 473.821,Z 626.88,A -85,B 0,C 180,E1 -7284.894,E2 -7284.894} C_VEL
LIN {X 0,Y 473.785,Z 630.298,A -85,B 0,C 180,E1 -7286.598,E2 -7286.598} C_VEL
LIN {X 0,Y 473.695,Z 632.317,A -85,B 0,C 180,E1 -7288.3,E2 -7288.3} C_VEL
LIN {X 0,Y 473.667,Z 632.985,A -85,B 0,C 180,E1 -7290,E2 -7290} C_VEL
LIN {X 0,Y 473.695,Z 632.315,A -85,B 0,C 180,E1 -7291.7,E2 -7291.7} C_VEL
LIN {X 0,Y 473.785,Z 630.296,A -85,B 0,C 180,E1 -7293.402,E2 -7293.402} C_VEL
LIN {X 0,Y 473.822,Z 626.877,A -85,B 0,C 180,E1 -7295.106,E2 -7295.106} C_VEL
LIN {X 0,Y 473.89,Z 621.959,A -85,B 0,C 180,E1 -7296.814,E2 -7296.814} C_VEL
LIN {X 0,Y 474.085,Z 615.401,A -85,B 0,C 180,E1 -7298.525,E2 -7298.525} C_VEL
LIN {X 0,Y 474.357,Z 608.112,A -85,B 0,C 180,E1 -7300.026,E2 -7300.026} C_VEL
LIN {X 0,Y 474.873,Z 599.099,A -85,B 0,C 180,E1 -7301.525,E2 -7301.525} C_VEL
LIN {X 0,Y 475.311,Z 589.648,A -85,B 0,C 180,E1 -7302.814,E2 -7302.814} C_VEL
LIN {X 0,Y 475.883,Z 579.2,A -85,B 0,C 180,E1 -7303.995,E2 -7303.995} C_VEL
LIN {X 0,Y 476.505,Z 567.686,A -85,B 0,C 180,E1 -7305.067,E2 -7305.067} C_VEL
LIN {X 0,Y 477.217,Z 554.938,A -85,B 0,C 180,E1 -7306.03,E2 -7306.03} C_VEL
LIN {X 0,Y 477.858,Z 541.657,A -85,B 0,C 180,E1 -7306.824,E2 -7306.824} C_VEL
LIN {X 0,Y 478.407,Z 528.372,A -85,B 0,C 180,E1 -7307.433,E2 -7307.433} C_VEL
LIN {X 0,Y 478.848,Z 514.585,A -85,B 0,C 180,E1 -7307.891,E2 -7307.891} C_VEL
LIN {X 0,Y 479.153,Z 500.476,A -85,B 0,C 180,E1 -7308.189,E2 -7308.189} C_VEL
LIN {X 0,Y 480.148,Z 389.802,A -85,B 0,C 180,E1 -7309.873,E2 -7309.873} C_VEL
LIN {X 0,Y 476.52,Z 369.356,A -85,B 0,C 180,E1 -7310.366,E2 -7310.366} C_VEL
LIN {X 0,Y 477.433,Z 350.207,A -85,B 0,C 180,E1 -7313.419,E2 -7313.419} C_VEL
LIN {X 0,Y 477.937,Z 340.367,A -85,B 0,C 180,E1 -7315.01,E2 -7315.01} C_VEL
LIN {X 0,Y 475.12,Z 326.877,A -85,B 0,C 180,E1 -7317.436,E2 -7317.436} C_VEL
LIN {X 0,Y 474.666,Z 324.984,A -85,B 0,C 180,E1 -7317.8,E2 -7317.8} C_VEL
LIN {X 0,Y 474.6,Z 324.99,A -85,B 0,C 180,E1 -7321.218,E2 -7321.218} C_VEL
LIN {X 0,Y 474.633,Z 324.988,A -85,B 0,C 180,E1 -7324.241,E2 -7324.241} C_VEL
LIN {X 0,Y 474.592,Z 324.99,A -85,B 0,C 180,E1 -7327.384,E2 -7327.384} C_VEL
LIN {X 0,Y 474.619,Z 324.991,A -85,B 0,C 180,E1 -7330.658,E2 -7330.658} C_VEL
LIN {X 0,Y 474.597,Z 324.987,A -85,B 0,C 180,E1 -7333.481,E2 -7333.481} C_VEL
LIN {X 0,Y 474.602,Z 324.994,A -85,B 0,C 180,E1 -7336.519,E2 -7336.519} C_VEL
LIN {X 0,Y 474.619,Z 324.985,A -85,B 0,C 180,E1 -7339.343,E2 -7339.343} C_VEL
LIN {X 0,Y 474.61,Z 324.986,A -85,B 0,C 180,E1 -7341.705,E2 -7341.705} C_VEL
LIN {X 0,Y 474.625,Z 324.988,A -85,B 0,C 180,E1 -7344.726,E2 -7344.726} C_VEL
LIN {X 0,Y 474.639,Z 324.984,A -85,B 0,C 180,E1 -7347.788,E2 -7347.788} C_VEL
LIN {X 0,Y 474.609,Z 324.987,A -85,B 0,C 180,E1 -7350.889,E2 -7350.889} C_VEL
LIN {X 0,Y 474.618,Z 324.985,A -85,B 0,C 180,E1 -7353.626,E2 -7353.626} C_VEL
LIN {X 0,Y 474.638,Z 324.984,A -85,B 0,C 180,E1 -7356.642,E2 -7356.642} C_VEL
LIN {X 0,Y 474.657,Z 324.988,A -85,B 0,C 180,E1 -7360.09,E2 -7360.09} C_VEL
LIN {X 0,Y 474.639,Z 324.982,A -85,B 0,C 180,E1 -7362.774,E2 -7362.774} C_VEL
LIN {X 0,Y 474.65,Z 324.982,A -85,B 0,C 180,E1 -7365.421,E2 -7365.421} C_VEL
LIN {X 0,Y 474.708,Z 324.978,A -85,B 0,C 180,E1 -7368.038,E2 -7368.038} C_VEL
LIN {X 0,Y 474.707,Z 324.974,A -85,B 0,C 180,E1 -7371.486,E2 -7371.486} C_VEL
LIN {X 0,Y 474.752,Z 324.976,A -85,B 0,C 180,E1 -7374.052,E2 -7374.052} C_VEL
LIN {X 0,Y 474.878,Z 324.95,A -85,B 0,C 180,E1 -7377.456,E2 -7377.456} C_VEL
LIN {X 0,Y 474.884,Z 324.957,A -85,B 0,C 180,E1 -7380,E2 -7380} C_VEL
LIN {X 0,Y 474.887,Z 324.951,A -85,B 0,C 180,E1 -7382.545,E2 -7382.545} C_VEL
LIN {X 0,Y 474.74,Z 324.971,A -85,B 0,C 180,E1 -7385.948,E2 -7385.948} C_VEL
LIN {X 0,Y 474.701,Z 324.976,A -85,B 0,C 180,E1 -7388.514,E2 -7388.514} C_VEL
LIN {X 0,Y 474.709,Z 324.977,A -85,B 0,C 180,E1 -7391.963,E2 -7391.963} C_VEL
LIN {X 0,Y 474.692,Z 324.981,A -85,B 0,C 180,E1 -7395.456,E2 -7395.456} C_VEL
LIN {X 0,Y 474.612,Z 324.988,A -85,B 0,C 180,E1 -7399.013,E2 -7399.013} C_VEL
LIN {X 0,Y 474.579,Z 324.996,A -85,B 0,C 180,E1 -7401.73,E2 -7401.73} C_VEL
LIN {X 0,Y 474.629,Z 324.981,A -85,B 0,C 180,E1 -7404.495,E2 -7404.495} C_VEL
LIN {X 0,Y 474.6,Z 324.993,A -85,B 0,C 180,E1 -7407.327,E2 -7407.327} C_VEL
LIN {X 0,Y 474.553,Z 324.981,A -85,B 0,C 180,E1 -7410.234,E2 -7410.234} C_VEL
LIN {X 0,Y 474.616,Z 324.989,A -85,B 0,C 180,E1 -7413.223,E2 -7413.223} C_VEL
LIN {X 0,Y 474.571,Z 324.981,A -85,B 0,C 180,E1 -7416.326,E2 -7416.326} C_VEL
LIN {X 0,Y 474.6,Z 324.992,A -85,B 0,C 180,E1 -7419.551,E2 -7419.551} C_VEL
LIN {X 0,Y 474.568,Z 324.995,A -85,B 0,C 180,E1 -7422.94,E2 -7422.94} C_VEL
LIN {X 0,Y 474.583,Z 324.99,A -85,B 0,C 180,E1 -7425.892,E2 -7425.892} C_VEL
LIN {X 0,Y 474.583,Z 324.995,A -85,B 0,C 180,E1 -7429.048,E2 -7429.048} C_VEL
LIN {X 0,Y 474.585,Z 324.995,A -85,B 0,C 180,E1 -7431.709,E2 -7431.709} C_VEL
LIN {X 0,Y 474.606,Z 324.991,A -85,B 0,C 180,E1 -7434.724,E2 -7434.724} C_VEL
LIN {X 0,Y 474.613,Z 324.989,A -85,B 0,C 180,E1 -7437.786,E2 -7437.786} C_VEL
LIN {X 0,Y 474.61,Z 325.131,A -85,B 0,C 180,E1 -7440.776,E2 -7440.776} C_VEL
LIN {X 0,Y 476.877,Z 336.225,A -85,B 0,C 180,E1 -7443.052,E2 -7443.052} C_VEL
LIN {X 0,Y 476.731,Z 343.116,A -85,B 0,C 180,E1 -7444.348,E2 -7444.348} C_VEL
LIN {X 0,Y 476.674,Z 344.93,A -85,B 0,C 180,E1 -7444.686,E2 -7444.686} C_VEL
LIN {X 0,Y 480.406,Z 362.617,A -85,B 0,C 180,E1 -7445.153,E2 -7445.153} C_VEL
LIN {X 0,Y 480.248,Z 374.814,A -85,B 0,C 180,E1 -7445.337,E2 -7445.337} C_VEL
LIN {X 0,Y 479.549,Z 380.666,A -85,B 0,C 180,E1 -7445.397,E2 -7445.397} C_VEL
LIN {X 0,Y 473.923,Z 399.703,A -85,B 0,C 180,E1 -7445.439,E2 -7445.439} C_VEL
LIN {X 0,Y 473.314,Z 405.55,A -85,B 0,C 180,E1 -7445.504,E2 -7445.504} C_VEL
LIN {X 0,Y 472.606,Z 481.759,A -85,B 0,C 180,E1 -7446.705,E2 -7446.705} C_VEL
LIN {X 0,Y 472.191,Z 495.798,A -85,B 0,C 180,E1 -7447.089,E2 -7447.089} C_VEL
LIN {X 0,Y 471.681,Z 509.263,A -85,B 0,C 180,E1 -7447.628,E2 -7447.628} C_VEL
LIN {X 0,Y 471.067,Z 522.397,A -85,B 0,C 180,E1 -7448.33,E2 -7448.33} C_VEL
LIN {X 0,Y 470.401,Z 535.307,A -85,B 0,C 180,E1 -7449.216,E2 -7449.216} C_VEL
LIN {X 0,Y 469.773,Z 546.825,A -85,B 0,C 180,E1 -7450.199,E2 -7450.199} C_VEL
LIN {X 0,Y 469.14,Z 556.694,A -85,B 0,C 180,E1 -7451.211,E2 -7451.211} C_VEL
LIN {X 0,Y 468.445,Z 567.419,A -85,B 0,C 180,E1 -7452.539,E2 -7452.539} C_VEL
LIN {X 0,Y 467.916,Z 577.064,A -85,B 0,C 180,E1 -7454.003,E2 -7454.003} C_VEL
LIN {X 0,Y 467.474,Z 584.657,A -85,B 0,C 180,E1 -7455.415,E2 -7455.415} C_VEL
LIN {X 0,Y 467.142,Z 591.383,A -85,B 0,C 180,E1 -7456.958,E2 -7456.958} C_VEL
LIN {X 0,Y 466.851,Z 597.318,A -85,B 0,C 180,E1 -7458.714,E2 -7458.714} C_VEL
LIN {X 0,Y 466.677,Z 601.651,A -85,B 0,C 180,E1 -7460.465,E2 -7460.465} C_VEL
LIN {X 0,Y 466.658,Z 604.518,A -85,B 0,C 180,E1 -7462.21,E2 -7462.21} C_VEL
LIN {X 0,Y 466.648,Z 606.013,A -85,B 0,C 180,E1 -7463.948,E2 -7463.948} C_VEL
LIN {X 0,Y 466.602,Z 606.182,A -85,B 0,C 180,E1 -7465.681,E2 -7465.681} C_VEL
LIN {X 0,Y 466.674,Z 605.032,A -85,B 0,C 180,E1 -7467.41,E2 -7467.41} C_VEL
LIN {X 0,Y 466.628,Z 602.558,A -85,B 0,C 180,E1 -7469.137,E2 -7469.137} C_VEL
LIN {X 0,Y 466.687,Z 598.673,A -85,B 0,C 180,E1 -7470.863,E2 -7470.863} C_VEL
LIN {X 0,Y 466.934,Z 593.245,A -85,B 0,C 180,E1 -7472.588,E2 -7472.588} C_VEL
LIN {X 0,Y 467.319,Z 588.105,A -85,B 0,C 180,E1 -7473.88,E2 -7473.88} C_VEL
LIN {X 0,Y 467.698,Z 580.712,A -85,B 0,C 180,E1 -7475.389,E2 -7475.389} C_VEL
LIN {X 0,Y 468.15,Z 573.021,A -85,B 0,C 180,E1 -7476.681,E2 -7476.681} C_VEL
LIN {X 0,Y 468.578,Z 563.425,A -85,B 0,C 180,E1 -7478.018,E2 -7478.018} C_VEL
LIN {X 0,Y 469.312,Z 552.485,A -85,B 0,C 180,E1 -7479.264,E2 -7479.264} C_VEL
LIN {X 0,Y 469.949,Z 541.001,A -85,B 0,C 180,E1 -7480.338,E2 -7480.338} C_VEL
LIN {X 0,Y 470.61,Z 528.26,A -85,B 0,C 180,E1 -7481.304,E2 -7481.304} C_VEL
LIN {X 0,Y 471.224,Z 515.799,A -85,B 0,C 180,E1 -7482.052,E2 -7482.052} C_VEL
LIN {X 0,Y 471.752,Z 503.191,A -85,B 0,C 180,E1 -7482.639,E2 -7482.639} C_VEL
LIN {X 0,Y 472.075,Z 489.081,A -85,B 0,C 180,E1 -7483.123,E2 -7483.123} C_VEL
LIN {X 0,Y 472.348,Z 475.532,A -85,B 0,C 180,E1 -7483.416,E2 -7483.416} C_VEL
LIN {X 0,Y 473.409,Z 362.874,A -85,B 0,C 180,E1 -7485.142,E2 -7485.142} C_VEL
LIN {X 0,Y 469.656,Z 345.093,A -85,B 0,C 180,E1 -7485.589,E2 -7485.589} C_VEL
LIN {X 0,Y 469.876,Z 337.372,A -85,B 0,C 180,E1 -7487.03,E2 -7487.03} C_VEL
LIN {X 0,Y 467.587,Z 325.87,A -85,B 0,C 180,E1 -7489.366,E2 -7489.366} C_VEL
LIN {X 0,Y 467.527,Z 325.873,A -85,B 0,C 180,E1 -7492.074,E2 -7492.074} C_VEL
LIN {X 0,Y 467.552,Z 325.874,A -85,B 0,C 180,E1 -7494.89,E2 -7494.89} C_VEL
LIN {X 0,Y 467.54,Z 325.869,A -85,B 0,C 180,E1 -7497.774,E2 -7497.774} C_VEL
LIN {X 0,Y 467.53,Z 325.875,A -85,B 0,C 180,E1 -7501.036,E2 -7501.036} C_VEL
LIN {X 0,Y 467.565,Z 325.866,A -85,B 0,C 180,E1 -7504.237,E2 -7504.237} C_VEL
LIN {X 0,Y 467.512,Z 325.874,A -85,B 0,C 180,E1 -7507.18,E2 -7507.18} C_VEL
LIN {X 0,Y 467.52,Z 325.872,A -85,B 0,C 180,E1 -7510.271,E2 -7510.271} C_VEL
LIN {X 0,Y 467.519,Z 325.874,A -85,B 0,C 180,E1 -7512.568,E2 -7512.568} C_VEL
LIN {X 0,Y 467.565,Z 325.866,A -85,B 0,C 180,E1 -7515.052,E2 -7515.052} C_VEL
